SPLINE
SPL {X  -133.930, Y  +759.019, Z    +0.000, E1   +46.142, E3 -160653.483}
SPL {X  -149.331, Y  +728.920, Z    +0.000, E1   +37.154, E3 -160670.653}
SPL {X  -155.856, Y  +707.636, Z    +0.000, E1   +27.210, E3 -160676.656}
SPL {X  -159.260, Y  +686.764, Z    +0.000, E1   +14.026, E3 -160679.931}
SPL {X  -159.985, Y  +672.780, Z    +0.000, E1    +3.059, E3 -160680.832}
SPL {X  -159.990, Y  +669.259, Z    +0.000, E1    -0.225, E3 -160680.888}
SPL {X  -159.990, Y  +665.054, Z    +0.000, E1    -7.292, E3 -160680.993}
SPL {X  -159.990, Y  +658.864, Z    +0.000, E1   -19.708, E3 -160681.381}
SPL {X  -159.990, Y  +650.462, Z    +0.000, E1   -35.240, E3 -160682.392}
SPL {X  -159.990, Y  +636.155, Z    +0.000, E1   -51.890, E3 -160685.290}
SPL {X  -159.990, Y  +583.574, Z    +0.000, E1   -66.740, E3 -160705.086}
SPL {X  -159.990, Y  +451.342, Z    +0.000, E1   -68.591, E3 -160790.778}
ENDSPLINE

SPLINE
SPL {X  -159.990, Y  +495.016, Z    +0.000, E1   -61.398, E3 -160804.742}
ENDSPLINE

SPLINE
SPL {X  -159.990, Y  +469.556, Z    +0.000, E1   -62.943, E3 -160822.182}
SPL {X  -159.990, Y  +452.168, Z    +0.000, E1   -63.738, E3 -160834.737}
SPL {X  -159.990, Y  +433.781, Z    +0.000, E1   -64.535, E3 -160847.762}
SPL {X  -159.990, Y  +407.091, Z    +0.000, E1   -65.705, E3 -160864.966}
SPL {X  -159.990, Y  +383.383, Z    +0.000, E1   -66.590, E3 -160880.100}
SPL {X  -159.086, Y  +365.512, Z    +0.000, E1   -67.201, E3 -160891.198}
SPL {X  -155.924, Y  +346.662, Z    +0.000, E1   -68.026, E3 -160900.715}
SPL {X  -152.004, Y  +332.585, Z    +0.000, E1   -68.049, E3 -160912.153}
SPL {X  -147.728, Y  +321.072, Z    +0.000, E1   -67.490, E3 -160925.735}
SPL {X  -142.939, Y  +310.631, Z    +0.000, E1   -66.808, E3 -160938.802}
SPL {X  -138.502, Y  +302.413, Z    +0.000, E1   -66.138, E3 -160949.544}
SPL {X  -133.815, Y  +294.806, Z    +0.000, E1   -65.413, E3 -160959.751}
SPL {X  -130.038, Y  +289.296, Z    +0.000, E1   -64.749, E3 -160967.342}
SPL {X  -127.114, Y  +285.347, Z    +0.000, E1   -64.250, E3 -160972.765}
SPL {X   -96.237, Y  +254.690, Z    +0.000, E1   -52.223, E3 -161116.153}
ENDSPLINE

SPLINE
SPL {X  -139.640, Y  +304.414, Z    +0.000, E1   -43.367, E3 -161236.514}
SPL {X  -151.122, Y  +329.974, Z    +0.000, E1   -34.701, E3 -161249.306}
SPL {X  -155.699, Y  +345.695, Z    +0.000, E1   -27.167, E3 -161253.687}
SPL {X  -158.589, Y  +361.372, Z    +0.000, E1   -17.765, E3 -161256.451}
SPL {X  -159.702, Y  +372.901, Z    +0.000, E1    -9.563, E3 -161257.683}
SPL {X  -159.980, Y  +380.731, Z    +0.000, E1    -3.359, E3 -161258.081}
SPL {X  -159.990, Y  +384.465, Z    +0.000, E1    -0.049, E3 -161258.138}
SPL {X  -159.990, Y  +385.295, Z    +0.000, E1    +1.130, E3 -161258.144}
SPL {X  -159.990, Y  +387.941, Z    +0.000, E1    +5.453, E3 -161258.208}
SPL {X  -159.990, Y  +392.683, Z    +0.000, E1   +14.335, E3 -161258.465}
SPL {X  -159.990, Y  +399.462, Z    +0.000, E1   +27.551, E3 -161259.151}
SPL {X  -159.990, Y  +406.707, Z    +0.000, E1   +39.277, E3 -161260.307}
SPL {X  -159.990, Y  +418.467, Z    +0.000, E1   +51.591, E3 -161262.913}
SPL {X  -159.990, Y  +469.047, Z    +0.000, E1   +66.225, E3 -161281.990}
SPL {X  -159.990, Y  +610.501, Z    +0.000, E1   +69.067, E3 -161369.594}
SPL {X  -159.990, Y  +630.690, Z    +0.000, E1   +69.080, E3 -161385.974}
SPL {X  -159.990, Y  +652.219, Z    +0.000, E1   +69.078, E3 -161403.459}
SPL {X  -159.990, Y  +671.254, Z    +0.000, E1   +69.063, E3 -161418.959}
SPL {X  -159.471, Y  +684.377, Z    +0.000, E1   +68.989, E3 -161430.187}
SPL {X  -158.115, Y  +695.924, Z    +0.000, E1   +68.836, E3 -161440.970}
SPL {X  -156.463, Y  +704.909, Z    +0.000, E1   +68.615, E3 -161450.028}
SPL {X  -154.598, Y  +712.687, Z    +0.000, E1   +68.393, E3 -161458.242}
SPL {X  -151.859, Y  +721.854, Z    +0.000, E1   +68.046, E3 -161468.461}
SPL {X  -148.628, Y  +730.715, Z    +0.000, E1   +67.614, E3 -161478.870}
SPL {X  -145.416, Y  +738.215, Z    +0.000, E1   +67.166, E3 -161488.078}
SPL {X  -141.128, Y  +746.863, Z    +0.000, E1   +66.582, E3 -161499.055}
SPL {X  -137.485, Y  +753.321, Z    +0.000, E1   +65.984, E3 -161507.632}
SPL {X  -134.819, Y  +757.643, Z    +0.000, E1   +65.575, E3 -161513.427}
SPL {X  -131.187, Y  +763.079, Z    +0.000, E1   +64.994, E3 -161520.810}
SPL {X  -127.405, Y  +768.272, Z    +0.000, E1   +64.349, E3 -161527.931}
SPL {X   -94.830, Y  +800.357, Z    +0.000, E1   +53.815, E3 -161642.463}
ENDSPLINE

SPLINE
SPL {X  -133.930, Y  +759.019, Z    +0.000, E1   +46.142, E3 -161789.846}
SPL {X  -149.331, Y  +728.920, Z    +0.000, E1   +37.154, E3 -161807.017}
SPL {X  -155.856, Y  +707.636, Z    +0.000, E1   +27.210, E3 -161813.020}
SPL {X  -158.677, Y  +691.955, Z    +0.000, E1   +17.570, E3 -161815.726}
SPL {X  -159.802, Y  +679.261, Z    +0.000, E1    +8.330, E3 -161816.922}
SPL {X  -159.990, Y  +669.767, Z    +0.000, E1    +0.394, E3 -161817.247}
SPL {X  -159.990, Y  +667.882, Z    +0.000, E1    -2.380, E3 -161817.269}
SPL {X  -159.990, Y  +664.041, Z    +0.000, E1    -9.423, E3 -161817.395}
SPL {X  -159.990, Y  +660.147, Z    +0.000, E1   -17.275, E3 -161817.632}
SPL {X  -159.990, Y  +656.649, Z    +0.000, E1   -24.355, E3 -161817.939}
SPL {X  -159.990, Y  +650.462, Z    +0.000, E1   -35.240, E3 -161818.756}
SPL {X  -159.990, Y  +636.155, Z    +0.000, E1   -51.890, E3 -161821.653}
SPL {X  -159.990, Y  +583.574, Z    +0.000, E1   -66.740, E3 -161841.450}
SPL {X  -159.990, Y  +451.342, Z    +0.000, E1   -68.591, E3 -161927.141}
ENDSPLINE

SPLINE
SPL {X  -159.990, Y  +495.016, Z    +0.000, E1   -61.398, E3 -161941.106}
ENDSPLINE

SPLINE
SPL {X  -159.990, Y  +469.556, Z    +0.000, E1   -62.943, E3 -161958.545}
SPL {X  -159.990, Y  +445.297, Z    +0.000, E1   -64.051, E3 -161976.035}
SPL {X  -159.990, Y  +420.812, Z    +0.000, E1   -65.111, E3 -161992.625}
SPL {X  -159.990, Y  +395.826, Z    +0.000, E1   -66.138, E3 -162008.561}
SPL {X  -159.536, Y  +370.459, Z    +0.000, E1   -67.052, E3 -162024.454}
SPL {X  -155.924, Y  +346.662, Z    +0.000, E1   -68.026, E3 -162037.079}
SPL {X  -152.004, Y  +332.585, Z    +0.000, E1   -68.049, E3 -162048.517}
SPL {X  -148.519, Y  +323.011, Z    +0.000, E1   -67.572, E3 -162059.794}
SPL {X  -144.736, Y  +314.321, Z    +0.000, E1   -67.058, E3 -162070.491}
SPL {X  -140.646, Y  +306.241, Z    +0.000, E1   -66.458, E3 -162080.870}
SPL {X  -136.388, Y  +298.863, Z    +0.000, E1   -65.814, E3 -162090.642}
SPL {X  -132.805, Y  +293.283, Z    +0.000, E1   -65.214, E3 -162098.232}
SPL {X  -130.038, Y  +289.296, Z    +0.000, E1   -64.749, E3 -162103.706}
SPL {X  -127.114, Y  +285.347, Z    +0.000, E1   -64.250, E3 -162109.129}
SPL {X   -96.237, Y  +254.690, Z    +0.000, E1   -52.223, E3 -162252.517}
ENDSPLINE

SPLINE
SPL {X  -139.640, Y  +304.414, Z    +0.000, E1   -43.367, E3 -162372.878}
SPL {X  -151.122, Y  +329.974, Z    +0.000, E1   -34.701, E3 -162385.670}
SPL {X  -155.699, Y  +345.695, Z    +0.000, E1   -27.167, E3 -162390.051}
SPL {X  -158.589, Y  +361.372, Z    +0.000, E1   -17.765, E3 -162392.815}
SPL {X  -159.702, Y  +372.901, Z    +0.000, E1    -9.563, E3 -162394.047}
SPL {X  -159.980, Y  +380.731, Z    +0.000, E1    -3.359, E3 -162394.445}
SPL {X  -159.990, Y  +384.465, Z    +0.000, E1    -0.049, E3 -162394.502}
SPL {X  -159.990, Y  +386.161, Z    +0.000, E1    +2.359, E3 -162394.525}
SPL {X  -159.990, Y  +391.786, Z    +0.000, E1   +12.382, E3 -162394.775}
SPL {X  -159.990, Y  +399.462, Z    +0.000, E1   +27.551, E3 -162395.515}
SPL {X  -159.990, Y  +406.707, Z    +0.000, E1   +39.277, E3 -162396.671}
SPL {X  -159.990, Y  +418.467, Z    +0.000, E1   +51.591, E3 -162399.276}
SPL {X  -159.990, Y  +469.047, Z    +0.000, E1   +66.225, E3 -162418.354}
SPL {X  -159.990, Y  +610.501, Z    +0.000, E1   +69.067, E3 -162505.957}
SPL {X  -159.990, Y  +623.913, Z    +0.000, E1   +69.046, E3 -162516.906}
SPL {X  -159.990, Y  +635.131, Z    +0.000, E1   +69.053, E3 -162526.007}
SPL {X  -159.990, Y  +652.219, Z    +0.000, E1   +69.078, E3 -162539.822}
SPL {X  -159.990, Y  +671.254, Z    +0.000, E1   +69.063, E3 -162555.323}
SPL {X  -159.471, Y  +684.377, Z    +0.000, E1   +68.989, E3 -162566.550}
SPL {X  -158.115, Y  +695.924, Z    +0.000, E1   +68.836, E3 -162577.334}
SPL {X  -156.463, Y  +704.909, Z    +0.000, E1   +68.615, E3 -162586.391}
SPL {X  -153.837, Y  +715.444, Z    +0.000, E1   +68.325, E3 -162597.569}
SPL {X  -151.088, Y  +724.124, Z    +0.000, E1   +67.925, E3 -162607.479}
SPL {X  -148.628, Y  +730.715, Z    +0.000, E1   +67.614, E3 -162615.234}
SPL {X  -145.416, Y  +738.215, Z    +0.000, E1   +67.166, E3 -162624.442}
SPL {X  -142.090, Y  +745.034, Z    +0.000, E1   +66.692, E3 -162633.098}
SPL {X  -138.343, Y  +751.861, Z    +0.000, E1   +66.137, E3 -162642.025}
SPL {X  -133.893, Y  +759.076, Z    +0.000, E1   +65.453, E3 -162651.701}
SPL {X  -130.341, Y  +764.280, Z    +0.000, E1   +64.831, E3 -162658.839}
SPL {X  -127.405, Y  +768.272, Z    +0.000, E1   +64.349, E3 -162664.294}
SPL {X   -94.830, Y  +800.357, Z    +0.000, E1   +53.815, E3 -162778.827}
ENDSPLINE

SPLINE
SPL {X  -133.930, Y  +759.019, Z    +0.000, E1   +46.142, E3 -162926.210}
SPL {X  -149.331, Y  +728.920, Z    +0.000, E1   +37.154, E3 -162943.381}
SPL {X  -155.856, Y  +707.636, Z    +0.000, E1   +27.210, E3 -162949.384}
SPL {X  -158.677, Y  +691.955, Z    +0.000, E1   +17.570, E3 -162952.090}
SPL {X  -159.802, Y  +679.261, Z    +0.000, E1    +8.330, E3 -162953.286}
SPL {X  -159.990, Y  +671.355, Z    +0.000, E1    +1.732, E3 -162953.596}
SPL {X  -159.990, Y  +669.259, Z    +0.000, E1    -0.225, E3 -162953.615}
SPL {X  -159.990, Y  +665.054, Z    +0.000, E1    -7.292, E3 -162953.720}
SPL {X  -159.990, Y  +658.864, Z    +0.000, E1   -19.708, E3 -162954.108}
SPL {X  -159.990, Y  +650.462, Z    +0.000, E1   -35.240, E3 -162955.120}
SPL {X  -159.990, Y  +636.155, Z    +0.000, E1   -51.890, E3 -162958.017}
SPL {X  -159.990, Y  +583.574, Z    +0.000, E1   -66.740, E3 -162977.813}
SPL {X  -159.990, Y  +451.342, Z    +0.000, E1   -68.591, E3 -163063.505}
ENDSPLINE

SPLINE
SPL {X  -159.990, Y  +495.016, Z    +0.000, E1   -61.398, E3 -163077.470}
ENDSPLINE

SPLINE
SPL {X  -159.990, Y  +473.575, Z    +0.000, E1   -62.704, E3 -163092.204}
SPL {X  -159.990, Y  +455.620, Z    +0.000, E1   -63.615, E3 -163104.822}
SPL {X  -159.990, Y  +433.781, Z    +0.000, E1   -64.535, E3 -163120.490}
SPL {X  -159.990, Y  +414.623, Z    +0.000, E1   -65.374, E3 -163132.910}
SPL {X  -159.990, Y  +395.826, Z    +0.000, E1   -66.138, E3 -163144.924}
SPL {X  -159.536, Y  +370.459, Z    +0.000, E1   -67.052, E3 -163160.817}
SPL {X  -155.924, Y  +346.662, Z    +0.000, E1   -68.026, E3 -163173.442}
SPL {X  -152.751, Y  +334.918, Z    +0.000, E1   -68.124, E3 -163182.272}
SPL {X  -150.185, Y  +327.353, Z    +0.000, E1   -67.790, E3 -163190.995}
SPL {X  -147.824, Y  +321.305, Z    +0.000, E1   -67.459, E3 -163198.258}
SPL {X  -144.736, Y  +314.321, Z    +0.000, E1   -67.058, E3 -163206.854}
SPL {X  -140.646, Y  +306.241, Z    +0.000, E1   -66.458, E3 -163217.233}
SPL {X  -137.570, Y  +300.823, Z    +0.000, E1   -65.968, E3 -163224.425}
SPL {X  -133.815, Y  +294.806, Z    +0.000, E1   -65.413, E3 -163232.478}
SPL {X  -130.038, Y  +289.296, Z    +0.000, E1   -64.749, E3 -163240.070}
SPL {X  -127.114, Y  +285.347, Z    +0.000, E1   -64.250, E3 -163245.493}
SPL {X   -96.237, Y  +254.690, Z    +0.000, E1   -52.223, E3 -163388.881}
ENDSPLINE

SPLINE
SPL {X  -139.640, Y  +304.414, Z    +0.000, E1   -43.367, E3 -163509.242}
SPL {X  -154.086, Y  +339.440, Z    +0.000, E1   -30.439, E3 -163524.799}
SPL {X  -158.589, Y  +361.372, Z    +0.000, E1   -17.765, E3 -163529.179}
SPL {X  -159.702, Y  +372.901, Z    +0.000, E1    -9.563, E3 -163530.411}
SPL {X  -159.980, Y  +380.731, Z    +0.000, E1    -3.359, E3 -163530.808}
SPL {X  -159.990, Y  +384.465, Z    +0.000, E1    -0.049, E3 -163530.866}
SPL {X  -159.990, Y  +386.161, Z    +0.000, E1    +2.359, E3 -163530.888}
SPL {X  -159.990, Y  +391.786, Z    +0.000, E1   +12.382, E3 -163531.139}
SPL {X  -159.990, Y  +399.462, Z    +0.000, E1   +27.551, E3 -163531.879}
SPL {X  -159.990, Y  +406.707, Z    +0.000, E1   +39.277, E3 -163533.034}
SPL {X  -159.990, Y  +418.467, Z    +0.000, E1   +51.591, E3 -163535.640}
SPL {X  -159.990, Y  +469.047, Z    +0.000, E1   +66.225, E3 -163554.717}
SPL {X  -159.990, Y  +610.501, Z    +0.000, E1   +69.067, E3 -163642.321}
SPL {X  -159.990, Y  +630.690, Z    +0.000, E1   +69.080, E3 -163658.701}
SPL {X  -159.990, Y  +648.088, Z    +0.000, E1   +69.056, E3 -163672.878}
SPL {X  -159.990, Y  +663.340, Z    +0.000, E1   +69.061, E3 -163685.264}
SPL {X  -159.706, Y  +681.022, Z    +0.000, E1   +69.040, E3 -163699.896}
SPL {X  -158.115, Y  +695.924, Z    +0.000, E1   +68.836, E3 -163713.697}
SPL {X  -156.463, Y  +704.909, Z    +0.000, E1   +68.615, E3 -163722.755}
SPL {X  -153.837, Y  +715.444, Z    +0.000, E1   +68.325, E3 -163733.932}
SPL {X  -151.088, Y  +724.124, Z    +0.000, E1   +67.925, E3 -163743.843}
SPL {X  -148.628, Y  +730.715, Z    +0.000, E1   +67.614, E3 -163751.597}
SPL {X  -145.416, Y  +738.215, Z    +0.000, E1   +67.166, E3 -163760.806}
SPL {X  -141.128, Y  +746.863, Z    +0.000, E1   +66.582, E3 -163771.783}
SPL {X  -137.485, Y  +753.321, Z    +0.000, E1   +65.984, E3 -163780.359}
SPL {X  -134.819, Y  +757.643, Z    +0.000, E1   +65.575, E3 -163786.154}
SPL {X  -131.187, Y  +763.079, Z    +0.000, E1   +64.994, E3 -163793.538}
SPL {X  -127.405, Y  +768.272, Z    +0.000, E1   +64.349, E3 -163800.658}
SPL {X   -94.830, Y  +800.357, Z    +0.000, E1   +53.815, E3 -163915.190}
ENDSPLINE

SPLINE
SPL {X  -133.930, Y  +759.019, Z    +0.000, E1   +46.142, E3 -164062.574}
SPL {X  -149.331, Y  +728.920, Z    +0.000, E1   +37.154, E3 -164079.744}
SPL {X  -155.856, Y  +707.636, Z    +0.000, E1   +27.210, E3 -164085.747}
SPL {X  -158.677, Y  +691.955, Z    +0.000, E1   +17.570, E3 -164088.453}
SPL {X  -159.802, Y  +679.261, Z    +0.000, E1    +8.330, E3 -164089.650}
SPL {X  -159.990, Y  +671.355, Z    +0.000, E1    +1.732, E3 -164089.960}
SPL {X  -159.990, Y  +669.500, Z    +0.000, E1    +0.000, E3 -164089.977}
SPL {X  -159.990, Y  +667.882, Z    +0.000, E1    -2.380, E3 -164089.996}
SPL {X  -159.990, Y  +664.041, Z    +0.000, E1    -9.423, E3 -164090.122}
SPL {X  -159.990, Y  +658.864, Z    +0.000, E1   -19.708, E3 -164090.472}
SPL {X  -159.990, Y  +650.462, Z    +0.000, E1   -35.240, E3 -164091.483}
SPL {X  -159.990, Y  +636.155, Z    +0.000, E1   -51.890, E3 -164094.381}
SPL {X  -159.990, Y  +583.574, Z    +0.000, E1   -66.740, E3 -164114.177}
SPL {X  -159.990, Y  +451.342, Z    +0.000, E1   -68.591, E3 -164199.869}
ENDSPLINE

SPLINE
SPL {X  -159.990, Y  +495.016, Z    +0.000, E1   -61.398, E3 -164213.833}
ENDSPLINE

SPLINE
SPL {X  -159.990, Y  +473.575, Z    +0.000, E1   -62.704, E3 -164228.568}
SPL {X  -159.990, Y  +455.620, Z    +0.000, E1   -63.615, E3 -164241.186}
SPL {X  -159.990, Y  +433.781, Z    +0.000, E1   -64.535, E3 -164256.853}
SPL {X  -159.990, Y  +407.091, Z    +0.000, E1   -65.705, E3 -164274.057}
SPL {X  -159.990, Y  +383.383, Z    +0.000, E1   -66.590, E3 -164289.191}
SPL {X  -158.268, Y  +359.089, Z    +0.000, E1   -67.514, E3 -164303.392}
SPL {X  -153.587, Y  +337.689, Z    +0.000, E1   -68.173, E3 -164316.126}
SPL {X  -150.185, Y  +327.353, Z    +0.000, E1   -67.790, E3 -164327.358}
SPL {X  -147.824, Y  +321.305, Z    +0.000, E1   -67.459, E3 -164334.622}
SPL {X  -144.736, Y  +314.321, Z    +0.000, E1   -67.058, E3 -164343.218}
SPL {X  -140.646, Y  +306.241, Z    +0.000, E1   -66.458, E3 -164353.597}
SPL {X  -136.388, Y  +298.863, Z    +0.000, E1   -65.814, E3 -164363.370}
SPL {X  -132.805, Y  +293.283, Z    +0.000, E1   -65.214, E3 -164370.959}
SPL {X  -130.038, Y  +289.296, Z    +0.000, E1   -64.749, E3 -164376.433}
SPL {X  -127.114, Y  +285.347, Z    +0.000, E1   -64.250, E3 -164381.856}
SPL {X   -96.237, Y  +254.690, Z    +0.000, E1   -52.223, E3 -164525.244}
ENDSPLINE

SPLINE
SPL {X  -139.640, Y  +304.414, Z    +0.000, E1   -43.367, E3 -164645.605}
SPL {X  -154.086, Y  +339.440, Z    +0.000, E1   -30.439, E3 -164661.162}
SPL {X  -158.589, Y  +361.372, Z    +0.000, E1   -17.765, E3 -164665.542}
SPL {X  -159.702, Y  +372.901, Z    +0.000, E1    -9.563, E3 -164666.774}
SPL {X  -159.980, Y  +380.731, Z    +0.000, E1    -3.359, E3 -164667.172}
SPL {X  -159.990, Y  +384.465, Z    +0.000, E1    -0.049, E3 -164667.229}
SPL {X  -159.990, Y  +386.161, Z    +0.000, E1    +2.359, E3 -164667.252}
SPL {X  -159.990, Y  +390.716, Z    +0.000, E1   +10.524, E3 -164667.427}
SPL {X  -159.990, Y  +397.792, Z    +0.000, E1   +24.215, E3 -164668.057}
SPL {X  -159.990, Y  +406.707, Z    +0.000, E1   +39.277, E3 -164669.398}
SPL {X  -159.990, Y  +418.467, Z    +0.000, E1   +51.591, E3 -164672.004}
SPL {X  -159.990, Y  +469.047, Z    +0.000, E1   +66.225, E3 -164691.081}
SPL {X  -159.990, Y  +610.501, Z    +0.000, E1   +69.067, E3 -164778.685}
SPL {X  -159.990, Y  +630.690, Z    +0.000, E1   +69.080, E3 -164795.065}
SPL {X  -159.990, Y  +652.219, Z    +0.000, E1   +69.078, E3 -164812.550}
SPL {X  -159.990, Y  +671.254, Z    +0.000, E1   +69.063, E3 -164828.050}
SPL {X  -159.172, Y  +687.655, Z    +0.000, E1   +68.973, E3 -164842.210}
SPL {X  -157.106, Y  +701.739, Z    +0.000, E1   +68.720, E3 -164855.818}
SPL {X  -153.837, Y  +715.444, Z    +0.000, E1   +68.325, E3 -164870.296}
SPL {X  -151.088, Y  +724.124, Z    +0.000, E1   +67.925, E3 -164880.206}
SPL {X  -148.628, Y  +730.715, Z    +0.000, E1   +67.614, E3 -164887.961}
SPL {X  -145.416, Y  +738.215, Z    +0.000, E1   +67.166, E3 -164897.169}
SPL {X  -142.090, Y  +745.034, Z    +0.000, E1   +66.692, E3 -164905.825}
SPL {X  -138.343, Y  +751.861, Z    +0.000, E1   +66.137, E3 -164914.752}
SPL {X  -133.893, Y  +759.076, Z    +0.000, E1   +65.453, E3 -164924.428}
SPL {X  -130.341, Y  +764.280, Z    +0.000, E1   +64.831, E3 -164931.566}
SPL {X  -127.405, Y  +768.272, Z    +0.000, E1   +64.349, E3 -164937.022}
SPL {X   -94.830, Y  +800.357, Z    +0.000, E1   +53.815, E3 -165051.554}
ENDSPLINE

SPLINE
SPL {X  -133.930, Y  +759.019, Z    +0.000, E1   +46.142, E3 -165198.937}
SPL {X  -149.331, Y  +728.920, Z    +0.000, E1   +37.154, E3 -165216.108}
SPL {X  -155.856, Y  +707.636, Z    +0.000, E1   +27.210, E3 -165222.111}
SPL {X  -158.677, Y  +691.955, Z    +0.000, E1   +17.570, E3 -165224.817}
SPL {X  -159.802, Y  +679.261, Z    +0.000, E1    +8.330, E3 -165226.013}
SPL {X  -159.990, Y  +669.483, Z    +0.000, E1    +0.154, E3 -165226.340}
SPL {X  -159.990, Y  +665.054, Z    +0.000, E1    -7.292, E3 -165226.447}
SPL {X  -159.990, Y  +660.147, Z    +0.000, E1   -17.275, E3 -165226.723}
SPL {X  -159.990, Y  +656.649, Z    +0.000, E1   -24.355, E3 -165227.030}
SPL {X  -159.990, Y  +650.462, Z    +0.000, E1   -35.240, E3 -165227.847}
SPL {X  -159.990, Y  +636.155, Z    +0.000, E1   -51.890, E3 -165230.744}
SPL {X  -159.990, Y  +583.574, Z    +0.000, E1   -66.740, E3 -165250.541}
SPL {X  -159.990, Y  +451.342, Z    +0.000, E1   -68.591, E3 -165336.232}
ENDSPLINE

SPLINE
SPL {X  -159.990, Y  +495.016, Z    +0.000, E1   -61.398, E3 -165350.197}
ENDSPLINE

SPLINE
SPL {X  -159.990, Y  +473.575, Z    +0.000, E1   -62.704, E3 -165364.932}
SPL {X  -159.990, Y  +455.620, Z    +0.000, E1   -63.615, E3 -165377.550}
SPL {X  -159.990, Y  +433.781, Z    +0.000, E1   -64.535, E3 -165393.217}
SPL {X  -159.990, Y  +414.623, Z    +0.000, E1   -65.374, E3 -165405.637}
SPL {X  -159.990, Y  +395.826, Z    +0.000, E1   -66.138, E3 -165417.652}
SPL {X  -159.536, Y  +370.459, Z    +0.000, E1   -67.052, E3 -165433.544}
SPL {X  -155.924, Y  +346.662, Z    +0.000, E1   -68.026, E3 -165446.170}
SPL {X  -152.751, Y  +334.918, Z    +0.000, E1   -68.124, E3 -165455.000}
SPL {X  -150.185, Y  +327.353, Z    +0.000, E1   -67.790, E3 -165463.722}
SPL {X  -147.824, Y  +321.305, Z    +0.000, E1   -67.459, E3 -165470.985}
SPL {X  -144.736, Y  +314.321, Z    +0.000, E1   -67.058, E3 -165479.582}
SPL {X  -140.646, Y  +306.241, Z    +0.000, E1   -66.458, E3 -165489.961}
SPL {X  -137.570, Y  +300.823, Z    +0.000, E1   -65.968, E3 -165497.152}
SPL {X  -133.815, Y  +294.806, Z    +0.000, E1   -65.413, E3 -165505.205}
SPL {X  -130.038, Y  +289.296, Z    +0.000, E1   -64.749, E3 -165512.797}
SPL {X  -127.114, Y  +285.347, Z    +0.000, E1   -64.250, E3 -165518.220}
SPL {X   -96.237, Y  +254.690, Z    +0.000, E1   -52.223, E3 -165661.608}
ENDSPLINE

SPLINE
SPL {X  -139.640, Y  +304.414, Z    +0.000, E1   -43.367, E3 -165781.969}
SPL {X  -154.086, Y  +339.440, Z    +0.000, E1   -30.439, E3 -165797.526}
SPL {X  -158.589, Y  +361.372, Z    +0.000, E1   -17.765, E3 -165801.906}
SPL {X  -159.702, Y  +372.901, Z    +0.000, E1    -9.563, E3 -165803.138}
SPL {X  -159.980, Y  +380.731, Z    +0.000, E1    -3.359, E3 -165803.536}
SPL {X  -159.990, Y  +384.708, Z    +0.000, E1    +0.166, E3 -165803.595}
SPL {X  -159.990, Y  +387.941, Z    +0.000, E1    +5.453, E3 -165803.662}
SPL {X  -159.990, Y  +391.582, Z    +0.000, E1   +12.331, E3 -165803.837}
SPL {X  -159.990, Y  +397.792, Z    +0.000, E1   +24.215, E3 -165804.421}
SPL {X  -159.990, Y  +406.707, Z    +0.000, E1   +39.277, E3 -165805.762}
SPL {X  -159.990, Y  +418.467, Z    +0.000, E1   +51.591, E3 -165808.367}
SPL {X  -159.990, Y  +469.047, Z    +0.000, E1   +66.225, E3 -165827.444}
SPL {X  -159.990, Y  +610.501, Z    +0.000, E1   +69.067, E3 -165915.048}
SPL {X  -159.990, Y  +630.690, Z    +0.000, E1   +69.080, E3 -165931.429}
SPL {X  -159.990, Y  +648.088, Z    +0.000, E1   +69.056, E3 -165945.605}
SPL {X  -159.990, Y  +663.340, Z    +0.000, E1   +69.061, E3 -165957.991}
SPL {X  -159.706, Y  +681.022, Z    +0.000, E1   +69.040, E3 -165972.624}
SPL {X  -158.115, Y  +695.924, Z    +0.000, E1   +68.836, E3 -165986.425}
SPL {X  -156.463, Y  +704.909, Z    +0.000, E1   +68.615, E3 -165995.482}
SPL {X  -153.837, Y  +715.444, Z    +0.000, E1   +68.325, E3 -166006.660}
SPL {X  -151.088, Y  +724.124, Z    +0.000, E1   +67.925, E3 -166016.570}
SPL {X  -148.628, Y  +730.715, Z    +0.000, E1   +67.614, E3 -166024.325}
SPL {X  -145.416, Y  +738.215, Z    +0.000, E1   +67.166, E3 -166033.533}
SPL {X  -142.090, Y  +745.034, Z    +0.000, E1   +66.692, E3 -166042.189}
SPL {X  -138.343, Y  +751.861, Z    +0.000, E1   +66.137, E3 -166051.115}
SPL {X  -133.893, Y  +759.076, Z    +0.000, E1   +65.453, E3 -166060.791}
SPL {X  -130.341, Y  +764.280, Z    +0.000, E1   +64.831, E3 -166067.930}
SPL {X  -127.405, Y  +768.272, Z    +0.000, E1   +64.349, E3 -166073.385}
SPL {X   -94.830, Y  +800.357, Z    +0.000, E1   +53.815, E3 -166187.917}
ENDSPLINE

SPLINE
SPL {X  -133.930, Y  +759.019, Z    +0.000, E1   +46.142, E3 -166335.301}
SPL {X  -149.331, Y  +728.920, Z    +0.000, E1   +37.154, E3 -166352.471}
SPL {X  -155.856, Y  +707.636, Z    +0.000, E1   +27.210, E3 -166358.475}
SPL {X  -159.260, Y  +686.764, Z    +0.000, E1   +14.026, E3 -166361.749}
SPL {X  -159.985, Y  +672.780, Z    +0.000, E1    +3.059, E3 -166362.650}
SPL {X  -159.990, Y  +669.259, Z    +0.000, E1    -0.225, E3 -166362.706}
SPL {X  -159.990, Y  +665.054, Z    +0.000, E1    -7.292, E3 -166362.811}
SPL {X  -159.990, Y  +658.864, Z    +0.000, E1   -19.708, E3 -166363.199}
SPL {X  -159.990, Y  +650.462, Z    +0.000, E1   -35.240, E3 -166364.211}
SPL {X  -159.990, Y  +636.155, Z    +0.000, E1   -51.890, E3 -166367.108}
SPL {X  -159.990, Y  +583.574, Z    +0.000, E1   -66.740, E3 -166386.904}
SPL {X  -159.990, Y  +451.342, Z    +0.000, E1   -68.591, E3 -166472.596}
ENDSPLINE

SPLINE
SPL {X  -159.990, Y  +495.016, Z    +0.000, E1   -61.398, E3 -166486.561}
ENDSPLINE

SPLINE
SPL {X  -159.990, Y  +469.556, Z    +0.000, E1   -62.943, E3 -166504.000}
SPL {X  -159.990, Y  +445.297, Z    +0.000, E1   -64.051, E3 -166521.489}
SPL {X  -159.990, Y  +420.812, Z    +0.000, E1   -65.111, E3 -166538.080}
SPL {X  -159.990, Y  +395.826, Z    +0.000, E1   -66.138, E3 -166554.015}
SPL {X  -159.536, Y  +370.459, Z    +0.000, E1   -67.052, E3 -166569.908}
SPL {X  -157.113, Y  +352.293, Z    +0.000, E1   -67.811, E3 -166579.490}
SPL {X  -153.587, Y  +337.689, Z    +0.000, E1   -68.173, E3 -166588.853}
SPL {X  -150.185, Y  +327.353, Z    +0.000, E1   -67.790, E3 -166600.086}
SPL {X  -147.050, Y  +319.468, Z    +0.000, E1   -67.370, E3 -166609.566}
SPL {X  -142.939, Y  +310.631, Z    +0.000, E1   -66.808, E3 -166620.620}
SPL {X  -138.502, Y  +302.413, Z    +0.000, E1   -66.138, E3 -166631.363}
SPL {X  -135.296, Y  +297.108, Z    +0.000, E1   -65.610, E3 -166638.502}
SPL {X  -132.805, Y  +293.283, Z    +0.000, E1   -65.214, E3 -166643.686}
SPL {X  -130.038, Y  +289.296, Z    +0.000, E1   -64.749, E3 -166649.160}
SPL {X  -127.114, Y  +285.347, Z    +0.000, E1   -64.250, E3 -166654.583}
SPL {X   -96.237, Y  +254.690, Z    +0.000, E1   -52.223, E3 -166797.972}
ENDSPLINE

SPLINE
SPL {X  -139.640, Y  +304.414, Z    +0.000, E1   -43.367, E3 -166918.332}
SPL {X  -154.086, Y  +339.440, Z    +0.000, E1   -30.439, E3 -166933.890}
SPL {X  -158.589, Y  +361.372, Z    +0.000, E1   -17.765, E3 -166938.270}
SPL {X  -159.702, Y  +372.901, Z    +0.000, E1    -9.563, E3 -166939.501}
SPL {X  -159.980, Y  +380.731, Z    +0.000, E1    -3.359, E3 -166939.899}
SPL {X  -159.990, Y  +384.465, Z    +0.000, E1    -0.049, E3 -166939.957}
SPL {X  -159.990, Y  +386.161, Z    +0.000, E1    +2.359, E3 -166939.979}
SPL {X  -159.990, Y  +391.786, Z    +0.000, E1   +12.382, E3 -166940.230}
SPL {X  -159.990, Y  +399.462, Z    +0.000, E1   +27.551, E3 -166940.970}
SPL {X  -159.990, Y  +406.707, Z    +0.000, E1   +39.277, E3 -166942.125}
SPL {X  -159.990, Y  +418.467, Z    +0.000, E1   +51.591, E3 -166944.731}
SPL {X  -159.990, Y  +469.047, Z    +0.000, E1   +66.225, E3 -166963.808}
SPL {X  -159.990, Y  +610.501, Z    +0.000, E1   +69.067, E3 -167051.412}
SPL {X  -159.990, Y  +630.690, Z    +0.000, E1   +69.080, E3 -167067.792}
SPL {X  -159.990, Y  +648.088, Z    +0.000, E1   +69.056, E3 -167081.969}
SPL {X  -159.990, Y  +663.340, Z    +0.000, E1   +69.061, E3 -167094.355}
SPL {X  -159.706, Y  +681.022, Z    +0.000, E1   +69.040, E3 -167108.987}
SPL {X  -158.115, Y  +695.924, Z    +0.000, E1   +68.836, E3 -167122.788}
SPL {X  -156.463, Y  +704.909, Z    +0.000, E1   +68.615, E3 -167131.846}
SPL {X  -153.837, Y  +715.444, Z    +0.000, E1   +68.325, E3 -167143.023}
SPL {X  -151.088, Y  +724.124, Z    +0.000, E1   +67.925, E3 -167152.933}
SPL {X  -148.628, Y  +730.715, Z    +0.000, E1   +67.614, E3 -167160.688}
SPL {X  -145.416, Y  +738.215, Z    +0.000, E1   +67.166, E3 -167169.897}
SPL {X  -141.128, Y  +746.863, Z    +0.000, E1   +66.582, E3 -167180.874}
SPL {X  -137.485, Y  +753.321, Z    +0.000, E1   +65.984, E3 -167189.450}
SPL {X  -134.819, Y  +757.643, Z    +0.000, E1   +65.575, E3 -167195.245}
SPL {X  -131.187, Y  +763.079, Z    +0.000, E1   +64.994, E3 -167202.628}
SPL {X  -127.405, Y  +768.272, Z    +0.000, E1   +64.349, E3 -167209.749}
SPL {X   -94.830, Y  +800.357, Z    +0.000, E1   +53.815, E3 -167324.281}
ENDSPLINE

SPLINE
SPL {X  -133.930, Y  +759.019, Z    +0.000, E1   +46.142, E3 -167471.665}
SPL {X  -149.331, Y  +728.920, Z    +0.000, E1   +37.154, E3 -167488.835}
SPL {X  -155.856, Y  +707.636, Z    +0.000, E1   +27.210, E3 -167494.838}
SPL {X  -158.677, Y  +691.955, Z    +0.000, E1   +17.570, E3 -167497.544}
SPL {X  -159.802, Y  +679.261, Z    +0.000, E1    +8.330, E3 -167498.741}
SPL {X  -159.990, Y  +671.355, Z    +0.000, E1    +1.732, E3 -167499.050}
SPL {X  -159.990, Y  +669.500, Z    +0.000, E1    +0.000, E3 -167499.068}
SPL {X  -159.990, Y  +667.882, Z    +0.000, E1    -2.380, E3 -167499.087}
SPL {X  -159.990, Y  +664.041, Z    +0.000, E1    -9.423, E3 -167499.213}
SPL {X  -159.990, Y  +658.864, Z    +0.000, E1   -19.708, E3 -167499.563}
SPL {X  -159.990, Y  +650.462, Z    +0.000, E1   -35.240, E3 -167500.574}
SPL {X  -159.990, Y  +636.155, Z    +0.000, E1   -51.890, E3 -167503.472}
SPL {X  -159.990, Y  +583.574, Z    +0.000, E1   -66.740, E3 -167523.268}
SPL {X  -159.990, Y  +451.342, Z    +0.000, E1   -68.591, E3 -167608.960}
ENDSPLINE

SPLINE
SPL {X  -159.990, Y  +501.364, Z    +0.000, E1   -60.990, E3 -167618.270}
ENDSPLINE

SPLINE
SPL {X  -159.990, Y  +489.357, Z    +0.000, E1   -61.712, E3 -167627.113}
SPL {X  -159.990, Y  +473.575, Z    +0.000, E1   -62.704, E3 -167637.659}
SPL {X  -159.990, Y  +455.620, Z    +0.000, E1   -63.615, E3 -167650.277}
SPL {X  -159.990, Y  +439.579, Z    +0.000, E1   -64.263, E3 -167662.012}
SPL {X  -159.990, Y  +420.812, Z    +0.000, E1   -65.111, E3 -167674.444}
SPL {X  -159.990, Y  +395.826, Z    +0.000, E1   -66.138, E3 -167690.379}
SPL {X  -159.536, Y  +370.459, Z    +0.000, E1   -67.052, E3 -167706.272}
SPL {X  -155.899, Y  +346.553, Z    +0.000, E1   -68.023, E3 -167719.018}
SPL {X  -155.470, Y  +344.740, Z    +0.000, E1   -66.275, E3 -167734.431}
SPL {X  -151.958, Y  +332.444, Z    +0.000, E1   -65.791, E3 -167749.177}
SPL {X  -148.012, Y  +321.760, Z    +0.000, E1   -65.212, E3 -167762.811}
SPL {X  -144.181, Y  +313.155, Z    +0.000, E1   -64.628, E3 -167774.320}
SPL {X  -141.300, Y  +307.460, Z    +0.000, E1   -64.150, E3 -167782.212}
SPL {X  -138.693, Y  +302.744, Z    +0.000, E1   -63.741, E3 -167788.826}
SPL {X  -135.031, Y  +296.690, Z    +0.000, E1   -63.147, E3 -167797.488}
SPL {X  -130.494, Y  +289.936, Z    +0.000, E1   -62.364, E3 -167807.326}
SPL {X  -102.192, Y  +259.400, Z    +0.000, E1   -52.167, E3 -167926.050}
ENDSPLINE

SPLINE
SPL {X  -140.725, Y  +306.386, Z    +0.000, E1   -41.058, E3 -168050.944}
SPL {X  -153.851, Y  +338.606, Z    +0.000, E1   -29.149, E3 -168067.561}
SPL {X  -158.264, Y  +359.064, Z    +0.000, E1   -18.155, E3 -168072.512}
SPL {X  -159.641, Y  +371.933, Z    +0.000, E1    -9.693, E3 -168074.247}
SPL {X  -159.986, Y  +381.420, Z    +0.000, E1    -2.704, E3 -168074.813}
SPL {X  -159.990, Y  +384.527, Z    +0.000, E1    +0.013, E3 -168074.873}
SPL {X  -159.990, Y  +386.984, Z    +0.000, E1    +3.187, E3 -168074.925}
SPL {X  -159.990, Y  +392.544, Z    +0.000, E1   +12.471, E3 -168075.238}
SPL {X  -159.990, Y  +397.827, Z    +0.000, E1   +22.184, E3 -168075.759}
SPL {X  -159.990, Y  +403.857, Z    +0.000, E1   +31.979, E3 -168076.723}
SPL {X  -159.990, Y  +417.858, Z    +0.000, E1   +47.695, E3 -168080.208}
SPL {X  -159.990, Y  +475.808, Z    +0.000, E1   +64.751, E3 -168104.162}
SPL {X  -159.990, Y  +590.266, Z    +0.000, E1   +66.680, E3 -168187.279}
SPL {X  -159.990, Y  +611.678, Z    +0.000, E1   +66.672, E3 -168206.919}
SPL {X  -159.990, Y  +629.811, Z    +0.000, E1   +66.653, E3 -168223.575}
SPL {X  -159.990, Y  +646.024, Z    +0.000, E1   +66.650, E3 -168238.451}
SPL {X  -159.990, Y  +658.527, Z    +0.000, E1   +66.634, E3 -168249.933}
SPL {X  -159.990, Y  +671.049, Z    +0.000, E1   +66.648, E3 -168261.382}
SPL {X  -159.584, Y  +682.893, Z    +0.000, E1   +66.583, E3 -168272.679}
SPL {X  -158.332, Y  +694.472, Z    +0.000, E1   +66.450, E3 -168284.553}
SPL {X  -156.148, Y  +706.350, Z    +0.000, E1   +66.133, E3 -168297.764}
SPL {X  -154.052, Y  +714.685, Z    +0.000, E1   +65.842, E3 -168307.551}
SPL {X  -151.974, Y  +721.507, Z    +0.000, E1   +65.548, E3 -168315.908}
SPL {X  -149.510, Y  +728.452, Z    +0.000, E1   +65.197, E3 -168324.751}
SPL {X  -145.784, Y  +737.407, Z    +0.000, E1   +64.671, E3 -168336.542}
SPL {X  -142.587, Y  +744.066, Z    +0.000, E1   +64.133, E3 -168345.725}
SPL {X  -139.326, Y  +750.145, Z    +0.000, E1   +63.650, E3 -168354.218}
SPL {X  -135.791, Y  +756.103, Z    +0.000, E1   +63.018, E3 -168362.863}
SPL {X  -133.172, Y  +760.168, Z    +0.000, E1   +62.565, E3 -168368.788}
SPL {X  -130.070, Y  +764.659, Z    +0.000, E1   +62.024, E3 -168375.383}
SPL {X  -103.420, Y  +793.570, Z    +0.000, E1   +51.337, E3 -168505.283}
ENDSPLINE

SPLINE
SPL {X  -132.256, Y  +761.529, Z    +0.000, E1   +44.935, E3 -168611.373}
SPL {X  -148.790, Y  +730.309, Z    +0.000, E1   +35.907, E3 -168632.646}
SPL {X  -157.132, Y  +701.603, Z    +0.000, E1   +22.438, E3 -168641.907}
SPL {X  -159.426, Y  +684.927, Z    +0.000, E1   +11.876, E3 -168644.526}
SPL {X  -159.929, Y  +675.915, Z    +0.000, E1    +5.290, E3 -168645.237}
SPL {X  -159.990, Y  +669.794, Z    +0.000, E1    +0.371, E3 -168645.410}
SPL {X  -159.990, Y  +668.338, Z    +0.000, E1    -1.468, E3 -168645.427}
SPL {X  -159.990, Y  +665.597, Z    +0.000, E1    -5.793, E3 -168645.505}
SPL {X  -159.990, Y  +662.769, Z    +0.000, E1   -10.720, E3 -168645.657}
SPL {X  -159.990, Y  +658.787, Z    +0.000, E1   -17.995, E3 -168645.985}
SPL {X  -159.990, Y  +653.215, Z    +0.000, E1   -27.908, E3 -168646.677}
SPL {X  -159.990, Y  +646.194, Z    +0.000, E1   -38.517, E3 -168647.965}
SPL {X  -159.990, Y  +636.314, Z    +0.000, E1   -48.490, E3 -168650.603}
SPL {X  -159.990, Y  +588.081, Z    +0.000, E1   -63.406, E3 -168671.785}
SPL {X  -159.990, Y  +471.514, Z    +0.000, E1   -66.231, E3 -168755.293}
SPL {X  -159.990, Y  +458.012, Z    +0.000, E1   -66.224, E3 -168767.922}
SPL {X  -159.990, Y  +445.900, Z    +0.000, E1   -66.225, E3 -168779.235}
ENDSPLINE

SPLINE
SPL {X  -159.990, Y  +468.953, Z    +0.000, E1   -61.697, E3 -168789.194}
ENDSPLINE

SPLINE
SPL {X  -159.990, Y  +457.098, Z    +0.000, E1   -61.912, E3 -168801.290}
SPL {X  -159.990, Y  +442.075, Z    +0.000, E1   -62.596, E3 -168813.066}
SPL {X  -159.990, Y  +430.868, Z    +0.000, E1   -63.135, E3 -168821.319}
SPL {X  -159.990, Y  +416.857, Z    +0.000, E1   -63.835, E3 -168830.986}
SPL {X  -159.990, Y  +402.942, Z    +0.000, E1   -64.377, E3 -168841.215}
SPL {X  -159.990, Y  +382.745, Z    +0.000, E1   -65.209, E3 -168855.129}
SPL {X  -158.929, Y  +364.101, Z    +0.000, E1   -65.981, E3 -168866.884}
SPL {X  -156.693, Y  +350.188, Z    +0.000, E1   -66.345, E3 -168877.008}
SPL {X  -154.578, Y  +341.238, Z    +0.000, E1   -66.113, E3 -168886.766}
SPL {X  -151.958, Y  +332.444, Z    +0.000, E1   -65.791, E3 -168897.326}
SPL {X  -148.012, Y  +321.760, Z    +0.000, E1   -65.212, E3 -168910.959}
SPL {X  -145.172, Y  +315.256, Z    +0.000, E1   -64.753, E3 -168919.664}
SPL {X  -142.205, Y  +309.188, Z    +0.000, E1   -64.322, E3 -168927.917}
SPL {X  -138.693, Y  +302.744, Z    +0.000, E1   -63.741, E3 -168936.974}
SPL {X  -135.977, Y  +298.197, Z    +0.000, E1   -63.280, E3 -168943.494}
SPL {X  -132.828, Y  +293.318, Z    +0.000, E1   -62.759, E3 -168950.548}
SPL {X  -129.451, Y  +288.482, Z    +0.000, E1   -62.137, E3 -168957.651}
SPL {X  -102.192, Y  +259.400, Z    +0.000, E1   -52.167, E3 -169074.198}
ENDSPLINE

SPLINE
SPL {X  -140.725, Y  +306.386, Z    +0.000, E1   -41.058, E3 -169199.092}
SPL {X  -153.851, Y  +338.606, Z    +0.000, E1   -29.149, E3 -169215.709}
SPL {X  -158.264, Y  +359.064, Z    +0.000, E1   -18.155, E3 -169220.660}
SPL {X  -159.641, Y  +371.933, Z    +0.000, E1    -9.693, E3 -169222.396}
SPL {X  -159.986, Y  +381.420, Z    +0.000, E1    -2.704, E3 -169222.961}
SPL {X  -159.990, Y  +384.527, Z    +0.000, E1    +0.013, E3 -169223.021}
SPL {X  -159.990, Y  +385.909, Z    +0.000, E1    +1.800, E3 -169223.039}
SPL {X  -159.990, Y  +389.230, Z    +0.000, E1    +6.815, E3 -169223.163}
SPL {X  -159.990, Y  +395.332, Z    +0.000, E1   +17.451, E3 -169223.646}
SPL {X  -159.990, Y  +403.857, Z    +0.000, E1   +31.979, E3 -169224.871}
SPL {X  -159.990, Y  +417.858, Z    +0.000, E1   +47.695, E3 -169228.356}
SPL {X  -159.990, Y  +475.808, Z    +0.000, E1   +64.751, E3 -169252.310}
SPL {X  -159.990, Y  +590.266, Z    +0.000, E1   +66.680, E3 -169335.427}
SPL {X  -159.990, Y  +605.903, Z    +0.000, E1   +66.635, E3 -169349.846}
SPL {X  -159.990, Y  +620.525, Z    +0.000, E1   +66.669, E3 -169363.180}
SPL {X  -159.990, Y  +638.202, Z    +0.000, E1   +66.649, E3 -169379.430}
SPL {X  -159.990, Y  +654.774, Z    +0.000, E1   +66.658, E3 -169394.599}
SPL {X  -159.990, Y  +671.049, Z    +0.000, E1   +66.648, E3 -169409.530}
SPL {X  -159.584, Y  +682.893, Z    +0.000, E1   +66.583, E3 -169420.827}
SPL {X  -158.845, Y  +690.607, Z    +0.000, E1   +66.486, E3 -169428.680}
SPL {X  -157.279, Y  +700.830, Z    +0.000, E1   +66.296, E3 -169439.661}
SPL {X  -154.589, Y  +712.719, Z    +0.000, E1   +65.941, E3 -169453.304}
SPL {X  -151.974, Y  +721.507, Z    +0.000, E1   +65.548, E3 -169464.056}
SPL {X  -149.510, Y  +728.452, Z    +0.000, E1   +65.197, E3 -169472.899}
SPL {X  -146.809, Y  +735.092, Z    +0.000, E1   +64.789, E3 -169481.646}
SPL {X  -143.550, Y  +742.141, Z    +0.000, E1   +64.312, E3 -169491.165}
SPL {X  -140.309, Y  +748.378, Z    +0.000, E1   +63.779, E3 -169499.898}
SPL {X  -136.621, Y  +754.755, Z    +0.000, E1   +63.190, E3 -169509.015}
SPL {X  -133.172, Y  +760.168, Z    +0.000, E1   +62.565, E3 -169516.936}
SPL {X  -130.070, Y  +764.659, Z    +0.000, E1   +62.024, E3 -169523.531}
SPL {X  -103.420, Y  +793.570, Z    +0.000, E1   +51.337, E3 -169653.431}
ENDSPLINE

SPLINE
SPL {X  -141.359, Y  +746.429, Z    +0.000, E1   +41.207, E3 -169771.645}
SPL {X  -153.791, Y  +715.605, Z    +0.000, E1   +29.700, E3 -169786.414}
SPL {X  -157.923, Y  +697.131, Z    +0.000, E1   +19.758, E3 -169790.946}
SPL {X  -159.426, Y  +684.927, Z    +0.000, E1   +11.876, E3 -169792.674}
SPL {X  -159.929, Y  +675.915, Z    +0.000, E1    +5.290, E3 -169793.385}
SPL {X  -159.990, Y  +669.794, Z    +0.000, E1    +0.371, E3 -169793.558}
SPL {X  -159.990, Y  +668.338, Z    +0.000, E1    -1.468, E3 -169793.575}
SPL {X  -159.990, Y  +664.217, Z    +0.000, E1    -7.944, E3 -169793.727}
SPL {X  -159.990, Y  +657.963, Z    +0.000, E1   -19.417, E3 -169794.224}
SPL {X  -159.990, Y  +649.570, Z    +0.000, E1   -33.681, E3 -169795.448}
SPL {X  -159.990, Y  +636.314, Z    +0.000, E1   -48.490, E3 -169798.751}
SPL {X  -159.990, Y  +588.081, Z    +0.000, E1   -63.406, E3 -169819.933}
SPL {X  -159.990, Y  +471.514, Z    +0.000, E1   -66.231, E3 -169903.441}
SPL {X  -159.990, Y  +458.012, Z    +0.000, E1   -66.224, E3 -169916.070}
SPL {X  -159.990, Y  +445.900, Z    +0.000, E1   -66.225, E3 -169927.383}
ENDSPLINE

SPLINE
SPL {X  -159.990, Y  +465.730, Z    +0.000, E1   -61.693, E3 -169941.208}
ENDSPLINE

SPLINE
SPL {X  -159.990, Y  +446.910, Z    +0.000, E1   -62.394, E3 -169957.428}
SPL {X  -159.990, Y  +430.868, Z    +0.000, E1   -63.135, E3 -169969.467}
SPL {X  -159.990, Y  +416.857, Z    +0.000, E1   -63.835, E3 -169979.134}
SPL {X  -159.990, Y  +402.942, Z    +0.000, E1   -64.377, E3 -169989.363}
SPL {X  -159.990, Y  +382.745, Z    +0.000, E1   -65.209, E3 -170003.277}
SPL {X  -158.342, Y  +359.598, Z    +0.000, E1   -66.150, E3 -170017.982}
SPL {X  -155.453, Y  +344.669, Z    +0.000, E1   -66.270, E3 -170030.824}
SPL {X  -151.958, Y  +332.444, Z    +0.000, E1   -65.791, E3 -170045.474}
SPL {X  -148.012, Y  +321.760, Z    +0.000, E1   -65.212, E3 -170059.107}
SPL {X  -144.181, Y  +313.155, Z    +0.000, E1   -64.628, E3 -170070.617}
SPL {X  -141.300, Y  +307.460, Z    +0.000, E1   -64.150, E3 -170078.508}
SPL {X  -138.693, Y  +302.744, Z    +0.000, E1   -63.741, E3 -170085.122}
SPL {X  -135.031, Y  +296.690, Z    +0.000, E1   -63.147, E3 -170093.784}
SPL {X  -130.494, Y  +289.936, Z    +0.000, E1   -62.364, E3 -170103.622}
SPL {X  -102.192, Y  +259.400, Z    +0.000, E1   -52.167, E3 -170222.346}
ENDSPLINE

SPLINE
SPL {X  -140.725, Y  +306.386, Z    +0.000, E1   -41.058, E3 -170347.240}
SPL {X  -153.851, Y  +338.606, Z    +0.000, E1   -29.149, E3 -170363.857}
SPL {X  -158.264, Y  +359.064, Z    +0.000, E1   -18.155, E3 -170368.809}
SPL {X  -159.641, Y  +371.933, Z    +0.000, E1    -9.693, E3 -170370.544}
SPL {X  -159.986, Y  +381.420, Z    +0.000, E1    -2.704, E3 -170371.109}
SPL {X  -159.990, Y  +384.527, Z    +0.000, E1    +0.013, E3 -170371.169}
SPL {X  -159.990, Y  +386.984, Z    +0.000, E1    +3.187, E3 -170371.221}
SPL {X  -159.990, Y  +390.572, Z    +0.000, E1    +9.243, E3 -170371.380}
SPL {X  -159.990, Y  +395.332, Z    +0.000, E1   +17.451, E3 -170371.794}
SPL {X  -159.990, Y  +403.857, Z    +0.000, E1   +31.979, E3 -170373.019}
SPL {X  -159.990, Y  +416.313, Z    +0.000, E1   +46.481, E3 -170376.012}
SPL {X  -159.990, Y  +425.447, Z    +0.000, E1   +52.896, E3 -170378.920}
SPL {X  -159.990, Y  +475.808, Z    +0.000, E1   +64.751, E3 -170400.458}
SPL {X  -159.990, Y  +586.159, Z    +0.000, E1   +66.648, E3 -170479.874}
SPL {X  -159.990, Y  +602.026, Z    +0.000, E1   +66.659, E3 -170494.391}
SPL {X  -159.990, Y  +615.972, Z    +0.000, E1   +66.639, E3 -170507.219}
SPL {X  -159.990, Y  +629.811, Z    +0.000, E1   +66.653, E3 -170519.871}
SPL {X  -159.990, Y  +646.024, Z    +0.000, E1   +66.650, E3 -170534.747}
SPL {X  -159.990, Y  +658.527, Z    +0.000, E1   +66.634, E3 -170546.229}
SPL {X  -159.990, Y  +671.049, Z    +0.000, E1   +66.648, E3 -170557.678}
SPL {X  -159.584, Y  +682.893, Z    +0.000, E1   +66.583, E3 -170568.976}
SPL {X  -158.332, Y  +694.472, Z    +0.000, E1   +66.450, E3 -170580.849}
SPL {X  -156.148, Y  +706.350, Z    +0.000, E1   +66.133, E3 -170594.061}
SPL {X  -154.052, Y  +714.685, Z    +0.000, E1   +65.842, E3 -170603.848}
SPL {X  -151.381, Y  +723.275, Z    +0.000, E1   +65.482, E3 -170614.395}
SPL {X  -147.622, Y  +733.180, Z    +0.000, E1   +64.943, E3 -170627.199}
SPL {X  -144.546, Y  +740.079, Z    +0.000, E1   +64.439, E3 -170636.527}
SPL {X  -141.166, Y  +746.792, Z    +0.000, E1   +63.950, E3 -170645.767}
SPL {X  -136.621, Y  +754.755, Z    +0.000, E1   +63.190, E3 -170657.163}
SPL {X  -133.172, Y  +760.168, Z    +0.000, E1   +62.565, E3 -170665.084}
SPL {X  -130.070, Y  +764.659, Z    +0.000, E1   +62.024, E3 -170671.680}
SPL {X  -103.420, Y  +793.570, Z    +0.000, E1   +51.337, E3 -170801.579}
ENDSPLINE

SPLINE
SPL {X  -141.359, Y  +746.429, Z    +0.000, E1   +41.207, E3 -170919.793}
SPL {X  -153.791, Y  +715.605, Z    +0.000, E1   +29.700, E3 -170934.562}
SPL {X  -157.923, Y  +697.131, Z    +0.000, E1   +19.758, E3 -170939.094}
SPL {X  -159.426, Y  +684.927, Z    +0.000, E1   +11.876, E3 -170940.823}
SPL {X  -159.972, Y  +673.894, Z    +0.000, E1    +3.783, E3 -170941.611}
SPL {X  -159.990, Y  +669.020, Z    +0.000, E1    -0.387, E3 -170941.715}
SPL {X  -159.990, Y  +664.217, Z    +0.000, E1    -7.944, E3 -170941.876}
SPL {X  -159.990, Y  +657.963, Z    +0.000, E1   -19.417, E3 -170942.372}
SPL {X  -159.990, Y  +649.570, Z    +0.000, E1   -33.681, E3 -170943.596}
SPL {X  -159.990, Y  +636.314, Z    +0.000, E1   -48.490, E3 -170946.900}
SPL {X  -159.990, Y  +588.081, Z    +0.000, E1   -63.406, E3 -170968.081}
SPL {X  -159.990, Y  +471.514, Z    +0.000, E1   -66.231, E3 -171051.589}
SPL {X  -159.990, Y  +458.012, Z    +0.000, E1   -66.224, E3 -171064.218}
SPL {X  -159.990, Y  +445.900, Z    +0.000, E1   -66.225, E3 -171075.532}
ENDSPLINE

SPLINE
SPL {X  -159.990, Y  +465.730, Z    +0.000, E1   -61.693, E3 -171089.356}
ENDSPLINE

SPLINE
SPL {X  -159.990, Y  +452.456, Z    +0.000, E1   -62.114, E3 -171101.284}
SPL {X  -159.990, Y  +436.367, Z    +0.000, E1   -62.893, E3 -171113.543}
SPL {X  -159.990, Y  +416.857, Z    +0.000, E1   -63.835, E3 -171127.282}
SPL {X  -159.990, Y  +397.192, Z    +0.000, E1   -64.622, E3 -171141.576}
SPL {X  -159.902, Y  +377.209, Z    +0.000, E1   -65.412, E3 -171155.140}
SPL {X  -158.342, Y  +359.598, Z    +0.000, E1   -66.150, E3 -171166.130}
SPL {X  -155.453, Y  +344.669, Z    +0.000, E1   -66.270, E3 -171178.972}
SPL {X  -152.827, Y  +335.165, Z    +0.000, E1   -65.880, E3 -171190.330}
SPL {X  -150.132, Y  +327.208, Z    +0.000, E1   -65.515, E3 -171200.223}
SPL {X  -147.311, Y  +320.081, Z    +0.000, E1   -65.083, E3 -171209.504}
SPL {X  -144.181, Y  +313.155, Z    +0.000, E1   -64.628, E3 -171218.765}
SPL {X  -141.300, Y  +307.460, Z    +0.000, E1   -64.150, E3 -171226.657}
SPL {X  -138.693, Y  +302.744, Z    +0.000, E1   -63.741, E3 -171233.271}
SPL {X  -135.031, Y  +296.690, Z    +0.000, E1   -63.147, E3 -171241.932}
SPL {X  -130.494, Y  +289.936, Z    +0.000, E1   -62.364, E3 -171251.770}
SPL {X  -102.192, Y  +259.400, Z    +0.000, E1   -52.167, E3 -171370.494}
ENDSPLINE

SPLINE
SPL {X  -140.725, Y  +306.386, Z    +0.000, E1   -41.058, E3 -171495.388}
SPL {X  -153.851, Y  +338.606, Z    +0.000, E1   -29.149, E3 -171512.006}
SPL {X  -158.264, Y  +359.064, Z    +0.000, E1   -18.155, E3 -171516.957}
SPL {X  -159.641, Y  +371.933, Z    +0.000, E1    -9.693, E3 -171518.692}
SPL {X  -159.986, Y  +381.420, Z    +0.000, E1    -2.704, E3 -171519.257}
SPL {X  -159.990, Y  +384.527, Z    +0.000, E1    +0.013, E3 -171519.318}
SPL {X  -159.990, Y  +385.909, Z    +0.000, E1    +1.800, E3 -171519.335}
SPL {X  -159.990, Y  +389.230, Z    +0.000, E1    +6.815, E3 -171519.459}
SPL {X  -159.990, Y  +395.332, Z    +0.000, E1   +17.451, E3 -171519.942}
SPL {X  -159.990, Y  +403.857, Z    +0.000, E1   +31.979, E3 -171521.167}
SPL {X  -159.990, Y  +417.858, Z    +0.000, E1   +47.695, E3 -171524.653}
SPL {X  -159.990, Y  +475.808, Z    +0.000, E1   +64.751, E3 -171548.606}
SPL {X  -159.990, Y  +586.159, Z    +0.000, E1   +66.648, E3 -171628.022}
SPL {X  -159.990, Y  +602.026, Z    +0.000, E1   +66.659, E3 -171642.539}
SPL {X  -159.990, Y  +620.525, Z    +0.000, E1   +66.669, E3 -171659.476}
SPL {X  -159.990, Y  +638.202, Z    +0.000, E1   +66.649, E3 -171675.726}
SPL {X  -159.990, Y  +654.774, Z    +0.000, E1   +66.658, E3 -171690.895}
SPL {X  -159.990, Y  +671.049, Z    +0.000, E1   +66.648, E3 -171705.826}
SPL {X  -159.230, Y  +687.071, Z    +0.000, E1   +66.569, E3 -171721.267}
SPL {X  -157.279, Y  +700.830, Z    +0.000, E1   +66.296, E3 -171735.957}
SPL {X  -154.589, Y  +712.719, Z    +0.000, E1   +65.941, E3 -171749.600}
SPL {X  -151.974, Y  +721.507, Z    +0.000, E1   +65.548, E3 -171760.353}
SPL {X  -149.510, Y  +728.452, Z    +0.000, E1   +65.197, E3 -171769.195}
SPL {X  -145.784, Y  +737.407, Z    +0.000, E1   +64.671, E3 -171780.986}
SPL {X  -142.587, Y  +744.066, Z    +0.000, E1   +64.133, E3 -171790.169}
SPL {X  -139.326, Y  +750.145, Z    +0.000, E1   +63.650, E3 -171798.662}
SPL {X  -135.791, Y  +756.103, Z    +0.000, E1   +63.018, E3 -171807.307}
SPL {X  -133.172, Y  +760.168, Z    +0.000, E1   +62.565, E3 -171813.232}
SPL {X  -130.070, Y  +764.659, Z    +0.000, E1   +62.024, E3 -171819.828}
SPL {X  -103.420, Y  +793.570, Z    +0.000, E1   +51.337, E3 -171949.727}
ENDSPLINE

SPLINE
SPL {X  -132.256, Y  +761.529, Z    +0.000, E1   +44.935, E3 -172055.817}
SPL {X  -148.790, Y  +730.309, Z    +0.000, E1   +35.907, E3 -172077.091}
SPL {X  -157.132, Y  +701.603, Z    +0.000, E1   +22.438, E3 -172086.352}
SPL {X  -159.426, Y  +684.927, Z    +0.000, E1   +11.876, E3 -172088.971}
SPL {X  -159.929, Y  +675.915, Z    +0.000, E1    +5.290, E3 -172089.681}
SPL {X  -159.990, Y  +669.794, Z    +0.000, E1    +0.371, E3 -172089.855}
SPL {X  -159.990, Y  +668.338, Z    +0.000, E1    -1.468, E3 -172089.871}
SPL {X  -159.990, Y  +665.597, Z    +0.000, E1    -5.793, E3 -172089.950}
SPL {X  -159.990, Y  +662.769, Z    +0.000, E1   -10.720, E3 -172090.101}
SPL {X  -159.990, Y  +658.787, Z    +0.000, E1   -17.995, E3 -172090.429}
SPL {X  -159.990, Y  +653.215, Z    +0.000, E1   -27.908, E3 -172091.121}
SPL {X  -159.990, Y  +646.194, Z    +0.000, E1   -38.517, E3 -172092.410}
SPL {X  -159.990, Y  +636.314, Z    +0.000, E1   -48.490, E3 -172095.048}
SPL {X  -159.990, Y  +588.081, Z    +0.000, E1   -63.406, E3 -172116.229}
SPL {X  -159.990, Y  +471.514, Z    +0.000, E1   -66.231, E3 -172199.737}
SPL {X  -159.990, Y  +458.012, Z    +0.000, E1   -66.224, E3 -172212.367}
SPL {X  -159.990, Y  +445.900, Z    +0.000, E1   -66.225, E3 -172223.680}
ENDSPLINE

SPLINE
SPL {X  -159.990, Y  +465.730, Z    +0.000, E1   -61.693, E3 -172237.504}
ENDSPLINE

SPLINE
SPL {X  -159.990, Y  +452.456, Z    +0.000, E1   -62.114, E3 -172249.432}
SPL {X  -159.990, Y  +436.367, Z    +0.000, E1   -62.893, E3 -172261.692}
SPL {X  -159.990, Y  +416.857, Z    +0.000, E1   -63.835, E3 -172275.431}
SPL {X  -159.990, Y  +397.192, Z    +0.000, E1   -64.622, E3 -172289.724}
SPL {X  -159.570, Y  +370.917, Z    +0.000, E1   -65.713, E3 -172307.081}
SPL {X  -156.693, Y  +350.188, Z    +0.000, E1   -66.345, E3 -172321.453}
SPL {X  -154.578, Y  +341.238, Z    +0.000, E1   -66.113, E3 -172331.211}
SPL {X  -151.958, Y  +332.444, Z    +0.000, E1   -65.791, E3 -172341.770}
SPL {X  -148.012, Y  +321.760, Z    +0.000, E1   -65.212, E3 -172355.404}
SPL {X  -144.181, Y  +313.155, Z    +0.000, E1   -64.628, E3 -172366.913}
SPL {X  -141.300, Y  +307.460, Z    +0.000, E1   -64.150, E3 -172374.805}
SPL {X  -138.693, Y  +302.744, Z    +0.000, E1   -63.741, E3 -172381.419}
SPL {X  -135.977, Y  +298.197, Z    +0.000, E1   -63.280, E3 -172387.939}
SPL {X  -132.828, Y  +293.318, Z    +0.000, E1   -62.759, E3 -172394.992}
SPL {X  -129.451, Y  +288.482, Z    +0.000, E1   -62.137, E3 -172402.096}
SPL {X  -102.192, Y  +259.400, Z    +0.000, E1   -52.167, E3 -172518.643}
ENDSPLINE

SPLINE
SPL {X  -140.725, Y  +306.386, Z    +0.000, E1   -41.058, E3 -172643.537}
SPL {X  -153.851, Y  +338.606, Z    +0.000, E1   -29.149, E3 -172660.154}
SPL {X  -157.523, Y  +354.512, Z    +0.000, E1   -20.811, E3 -172664.280}
SPL {X  -159.458, Y  +369.460, Z    +0.000, E1   -11.469, E3 -172666.569}
SPL {X  -159.986, Y  +381.420, Z    +0.000, E1    -2.704, E3 -172667.405}
SPL {X  -159.990, Y  +384.527, Z    +0.000, E1    +0.013, E3 -172667.466}
SPL {X  -159.990, Y  +385.909, Z    +0.000, E1    +1.800, E3 -172667.483}
SPL {X  -159.990, Y  +389.230, Z    +0.000, E1    +6.815, E3 -172667.608}
SPL {X  -159.990, Y  +395.332, Z    +0.000, E1   +17.451, E3 -172668.090}
SPL {X  -159.990, Y  +403.857, Z    +0.000, E1   +31.979, E3 -172669.316}
SPL {X  -159.990, Y  +417.858, Z    +0.000, E1   +47.695, E3 -172672.801}
SPL {X  -159.990, Y  +475.808, Z    +0.000, E1   +64.751, E3 -172696.754}
SPL {X  -159.990, Y  +590.266, Z    +0.000, E1   +66.680, E3 -172779.872}
SPL {X  -159.990, Y  +611.678, Z    +0.000, E1   +66.672, E3 -172799.511}
SPL {X  -159.990, Y  +625.813, Z    +0.000, E1   +66.632, E3 -172812.543}
SPL {X  -159.990, Y  +638.202, Z    +0.000, E1   +66.649, E3 -172823.874}
SPL {X  -159.990, Y  +654.774, Z    +0.000, E1   +66.658, E3 -172839.043}
SPL {X  -159.990, Y  +671.049, Z    +0.000, E1   +66.648, E3 -172853.974}
SPL {X  -159.584, Y  +682.893, Z    +0.000, E1   +66.583, E3 -172865.272}
SPL {X  -158.332, Y  +694.472, Z    +0.000, E1   +66.450, E3 -172877.145}
SPL {X  -156.148, Y  +706.350, Z    +0.000, E1   +66.133, E3 -172890.357}
SPL {X  -154.052, Y  +714.685, Z    +0.000, E1   +65.842, E3 -172900.144}
SPL {X  -151.381, Y  +723.275, Z    +0.000, E1   +65.482, E3 -172910.691}
SPL {X  -147.622, Y  +733.180, Z    +0.000, E1   +64.943, E3 -172923.495}
SPL {X  -144.546, Y  +740.079, Z    +0.000, E1   +64.439, E3 -172932.823}
SPL {X  -142.587, Y  +744.066, Z    +0.000, E1   +64.133, E3 -172938.317}
SPL {X  -139.326, Y  +750.145, Z    +0.000, E1   +63.650, E3 -172946.810}
SPL {X  -135.791, Y  +756.103, Z    +0.000, E1   +63.018, E3 -172955.456}
SPL {X  -133.172, Y  +760.168, Z    +0.000, E1   +62.565, E3 -172961.380}
SPL {X  -130.070, Y  +764.659, Z    +0.000, E1   +62.024, E3 -172967.976}
SPL {X  -103.420, Y  +793.570, Z    +0.000, E1   +51.337, E3 -173097.876}
ENDSPLINE

SPLINE
SPL {X  -132.256, Y  +761.529, Z    +0.000, E1   +44.935, E3 -173203.965}
SPL {X  -148.790, Y  +730.309, Z    +0.000, E1   +35.907, E3 -173225.239}
SPL {X  -157.132, Y  +701.603, Z    +0.000, E1   +22.438, E3 -173234.500}
SPL {X  -159.426, Y  +684.927, Z    +0.000, E1   +11.876, E3 -173237.119}
SPL {X  -159.972, Y  +673.894, Z    +0.000, E1    +3.783, E3 -173237.907}
SPL {X  -159.990, Y  +669.020, Z    +0.000, E1    -0.387, E3 -173238.012}
SPL {X  -159.990, Y  +664.217, Z    +0.000, E1    -7.944, E3 -173238.172}
SPL {X  -159.990, Y  +657.963, Z    +0.000, E1   -19.417, E3 -173238.669}
SPL {X  -159.990, Y  +649.570, Z    +0.000, E1   -33.681, E3 -173239.893}
SPL {X  -159.990, Y  +636.314, Z    +0.000, E1   -48.490, E3 -173243.196}
SPL {X  -159.990, Y  +588.081, Z    +0.000, E1   -63.406, E3 -173264.377}
SPL {X  -159.990, Y  +471.514, Z    +0.000, E1   -66.231, E3 -173347.885}
SPL {X  -159.990, Y  +458.012, Z    +0.000, E1   -66.224, E3 -173360.515}
SPL {X  -159.990, Y  +445.900, Z    +0.000, E1   -66.225, E3 -173371.828}
ENDSPLINE

SPLINE
SPL {X  -159.990, Y  +468.953, Z    +0.000, E1   -61.697, E3 -173381.786}
ENDSPLINE

SPLINE
SPL {X  -159.990, Y  +457.098, Z    +0.000, E1   -61.912, E3 -173393.883}
SPL {X  -159.990, Y  +442.075, Z    +0.000, E1   -62.596, E3 -173405.658}
SPL {X  -159.990, Y  +430.868, Z    +0.000, E1   -63.135, E3 -173413.912}
SPL {X  -159.990, Y  +416.857, Z    +0.000, E1   -63.835, E3 -173423.579}
SPL {X  -159.990, Y  +397.192, Z    +0.000, E1   -64.622, E3 -173437.872}
SPL {X  -159.570, Y  +370.917, Z    +0.000, E1   -65.713, E3 -173455.229}
SPL {X  -156.693, Y  +350.188, Z    +0.000, E1   -66.345, E3 -173469.601}
SPL {X  -153.533, Y  +337.508, Z    +0.000, E1   -66.008, E3 -173483.733}
SPL {X  -150.132, Y  +327.208, Z    +0.000, E1   -65.515, E3 -173496.519}
SPL {X  -146.325, Y  +317.802, Z    +0.000, E1   -64.967, E3 -173508.774}
SPL {X  -142.205, Y  +309.188, Z    +0.000, E1   -64.322, E3 -173520.510}
SPL {X  -138.693, Y  +302.744, Z    +0.000, E1   -63.741, E3 -173529.567}
SPL {X  -135.031, Y  +296.690, Z    +0.000, E1   -63.147, E3 -173538.228}
SPL {X  -130.494, Y  +289.936, Z    +0.000, E1   -62.364, E3 -173548.066}
SPL {X  -102.192, Y  +259.400, Z    +0.000, E1   -52.167, E3 -173666.791}
ENDSPLINE

SPLINE
SPL {X  -140.725, Y  +306.386, Z    +0.000, E1   -41.058, E3 -173791.685}
SPL {X  -153.851, Y  +338.606, Z    +0.000, E1   -29.149, E3 -173808.302}
SPL {X  -157.523, Y  +354.512, Z    +0.000, E1   -20.811, E3 -173812.428}
SPL {X  -159.458, Y  +369.460, Z    +0.000, E1   -11.469, E3 -173814.718}
SPL {X  -159.986, Y  +381.420, Z    +0.000, E1    -2.704, E3 -173815.553}
SPL {X  -159.990, Y  +385.016, Z    +0.000, E1    +0.442, E3 -173815.620}
SPL {X  -159.990, Y  +389.230, Z    +0.000, E1    +6.815, E3 -173815.756}
SPL {X  -159.990, Y  +393.768, Z    +0.000, E1   +14.836, E3 -173816.074}
SPL {X  -159.990, Y  +397.827, Z    +0.000, E1   +22.184, E3 -173816.500}
SPL {X  -159.990, Y  +403.857, Z    +0.000, E1   +31.979, E3 -173817.464}
SPL {X  -159.990, Y  +417.858, Z    +0.000, E1   +47.695, E3 -173820.949}
SPL {X  -159.990, Y  +475.808, Z    +0.000, E1   +64.751, E3 -173844.902}
SPL {X  -159.990, Y  +590.266, Z    +0.000, E1   +66.680, E3 -173928.020}
SPL {X  -159.990, Y  +605.903, Z    +0.000, E1   +66.635, E3 -173942.439}
SPL {X  -159.990, Y  +620.525, Z    +0.000, E1   +66.669, E3 -173955.773}
SPL {X  -159.990, Y  +638.202, Z    +0.000, E1   +66.649, E3 -173972.022}
SPL {X  -159.990, Y  +649.814, Z    +0.000, E1   +66.629, E3 -173982.710}
SPL {X  -159.990, Y  +658.527, Z    +0.000, E1   +66.634, E3 -173990.673}
SPL {X  -159.990, Y  +671.049, Z    +0.000, E1   +66.648, E3 -174002.122}
SPL {X  -159.584, Y  +682.893, Z    +0.000, E1   +66.583, E3 -174013.420}
SPL {X  -158.332, Y  +694.472, Z    +0.000, E1   +66.450, E3 -174025.294}
SPL {X  -156.148, Y  +706.350, Z    +0.000, E1   +66.133, E3 -174038.505}
SPL {X  -154.052, Y  +714.685, Z    +0.000, E1   +65.842, E3 -174048.292}
SPL {X  -151.974, Y  +721.507, Z    +0.000, E1   +65.548, E3 -174056.649}
SPL {X  -149.510, Y  +728.452, Z    +0.000, E1   +65.197, E3 -174065.492}
SPL {X  -146.809, Y  +735.092, Z    +0.000, E1   +64.789, E3 -174074.239}
SPL {X  -143.550, Y  +742.141, Z    +0.000, E1   +64.312, E3 -174083.757}
SPL {X  -140.309, Y  +748.378, Z    +0.000, E1   +63.779, E3 -174092.490}
SPL {X  -136.621, Y  +754.755, Z    +0.000, E1   +63.190, E3 -174101.607}
SPL {X  -133.172, Y  +760.168, Z    +0.000, E1   +62.565, E3 -174109.528}
SPL {X  -130.070, Y  +764.659, Z    +0.000, E1   +62.024, E3 -174116.124}
SPL {X  -103.420, Y  +793.570, Z    +0.000, E1   +51.337, E3 -174246.024}
ENDSPLINE

SPLINE
SPL {X  -132.256, Y  +761.529, Z    +0.000, E1   +44.935, E3 -174352.113}
SPL {X  -148.790, Y  +730.309, Z    +0.000, E1   +35.907, E3 -174373.387}
SPL {X  -157.132, Y  +701.603, Z    +0.000, E1   +22.438, E3 -174382.648}
SPL {X  -159.426, Y  +684.927, Z    +0.000, E1   +11.876, E3 -174385.267}
SPL {X  -159.929, Y  +675.915, Z    +0.000, E1    +5.290, E3 -174385.977}
SPL {X  -159.990, Y  +669.794, Z    +0.000, E1    +0.371, E3 -174386.151}
SPL {X  -159.990, Y  +668.338, Z    +0.000, E1    -1.468, E3 -174386.168}
SPL {X  -159.990, Y  +664.217, Z    +0.000, E1    -7.944, E3 -174386.320}
SPL {X  -159.990, Y  +658.787, Z    +0.000, E1   -17.995, E3 -174386.725}
SPL {X  -159.990, Y  +653.215, Z    +0.000, E1   -27.908, E3 -174387.417}
SPL {X  -159.990, Y  +646.194, Z    +0.000, E1   -38.517, E3 -174388.706}
SPL {X  -159.990, Y  +636.314, Z    +0.000, E1   -48.490, E3 -174391.344}
SPL {X  -159.990, Y  +588.081, Z    +0.000, E1   -63.406, E3 -174412.525}
SPL {X  -159.990, Y  +471.514, Z    +0.000, E1   -66.231, E3 -174496.033}
SPL {X  -159.990, Y  +458.012, Z    +0.000, E1   -66.224, E3 -174508.663}
SPL {X  -159.990, Y  +445.900, Z    +0.000, E1   -66.225, E3 -174519.976}
ENDSPLINE

SPLINE
SPL {X  -159.990, Y  +465.730, Z    +0.000, E1   -61.693, E3 -174533.801}
ENDSPLINE

SPLINE
SPL {X  -159.990, Y  +452.456, Z    +0.000, E1   -62.114, E3 -174545.728}
SPL {X  -159.990, Y  +436.367, Z    +0.000, E1   -62.893, E3 -174557.988}
SPL {X  -159.990, Y  +416.857, Z    +0.000, E1   -63.835, E3 -174571.727}
SPL {X  -159.990, Y  +397.192, Z    +0.000, E1   -64.622, E3 -174586.020}
SPL {X  -159.902, Y  +377.209, Z    +0.000, E1   -65.412, E3 -174599.584}
SPL {X  -158.342, Y  +359.598, Z    +0.000, E1   -66.150, E3 -174610.575}
SPL {X  -155.453, Y  +344.669, Z    +0.000, E1   -66.270, E3 -174623.417}
SPL {X  -152.827, Y  +335.165, Z    +0.000, E1   -65.880, E3 -174634.774}
SPL {X  -150.132, Y  +327.208, Z    +0.000, E1   -65.515, E3 -174644.667}
SPL {X  -147.311, Y  +320.081, Z    +0.000, E1   -65.083, E3 -174653.948}
SPL {X  -144.181, Y  +313.155, Z    +0.000, E1   -64.628, E3 -174663.209}
SPL {X  -141.300, Y  +307.460, Z    +0.000, E1   -64.150, E3 -174671.101}
SPL {X  -138.693, Y  +302.744, Z    +0.000, E1   -63.741, E3 -174677.715}
SPL {X  -135.977, Y  +298.197, Z    +0.000, E1   -63.280, E3 -174684.235}
SPL {X  -132.828, Y  +293.318, Z    +0.000, E1   -62.759, E3 -174691.288}
SPL {X  -129.451, Y  +288.482, Z    +0.000, E1   -62.137, E3 -174698.392}
SPL {X  -102.192, Y  +259.400, Z    +0.000, E1   -52.167, E3 -174814.939}
ENDSPLINE

SPLINE
SPL {X  -140.725, Y  +306.386, Z    +0.000, E1   -41.058, E3 -174939.833}
SPL {X  -153.851, Y  +338.606, Z    +0.000, E1   -29.149, E3 -174956.450}
SPL {X  -158.264, Y  +359.064, Z    +0.000, E1   -18.155, E3 -174961.401}
SPL {X  -159.641, Y  +371.933, Z    +0.000, E1    -9.693, E3 -174963.136}
SPL {X  -159.986, Y  +381.420, Z    +0.000, E1    -2.704, E3 -174963.701}
SPL {X  -159.990, Y  +384.527, Z    +0.000, E1    +0.013, E3 -174963.762}
SPL {X  -159.990, Y  +385.909, Z    +0.000, E1    +1.800, E3 -174963.779}
SPL {X  -159.990, Y  +389.230, Z    +0.000, E1    +6.815, E3 -174963.904}
SPL {X  -159.990, Y  +395.332, Z    +0.000, E1   +17.451, E3 -174964.387}
SPL {X  -159.990, Y  +403.857, Z    +0.000, E1   +31.979, E3 -174965.612}
SPL {X  -159.990, Y  +417.858, Z    +0.000, E1   +47.695, E3 -174969.097}
SPL {X  -159.990, Y  +475.808, Z    +0.000, E1   +64.751, E3 -174993.051}
SPL {X  -159.990, Y  +586.159, Z    +0.000, E1   +66.648, E3 -175072.467}
SPL {X  -159.990, Y  +602.026, Z    +0.000, E1   +66.659, E3 -175086.983}
SPL {X  -159.990, Y  +620.525, Z    +0.000, E1   +66.669, E3 -175103.921}
SPL {X  -159.990, Y  +638.202, Z    +0.000, E1   +66.649, E3 -175120.171}
SPL {X  -159.990, Y  +654.774, Z    +0.000, E1   +66.658, E3 -175135.340}
SPL {X  -159.990, Y  +671.049, Z    +0.000, E1   +66.648, E3 -175150.270}
SPL {X  -159.230, Y  +687.071, Z    +0.000, E1   +66.569, E3 -175165.712}
SPL {X  -157.279, Y  +700.830, Z    +0.000, E1   +66.296, E3 -175180.402}
SPL {X  -154.589, Y  +712.719, Z    +0.000, E1   +65.941, E3 -175194.045}
SPL {X  -151.381, Y  +723.275, Z    +0.000, E1   +65.482, E3 -175206.988}
SPL {X  -147.622, Y  +733.180, Z    +0.000, E1   +64.943, E3 -175219.791}
SPL {X  -143.550, Y  +742.141, Z    +0.000, E1   +64.312, E3 -175231.905}
SPL {X  -139.326, Y  +750.145, Z    +0.000, E1   +63.650, E3 -175243.107}
SPL {X  -135.791, Y  +756.103, Z    +0.000, E1   +63.018, E3 -175251.752}
SPL {X  -133.172, Y  +760.168, Z    +0.000, E1   +62.565, E3 -175257.677}
SPL {X  -130.070, Y  +764.659, Z    +0.000, E1   +62.024, E3 -175264.272}
SPL {X  -103.420, Y  +793.570, Z    +0.000, E1   +51.337, E3 -175394.172}
ENDSPLINE

SPLINE
SPL {X  -141.359, Y  +746.429, Z    +0.000, E1   +41.207, E3 -175512.386}
SPL {X  -153.791, Y  +715.605, Z    +0.000, E1   +29.700, E3 -175527.155}
SPL {X  -157.923, Y  +697.131, Z    +0.000, E1   +19.758, E3 -175531.686}
SPL {X  -159.426, Y  +684.927, Z    +0.000, E1   +11.876, E3 -175533.415}
SPL {X  -159.972, Y  +673.894, Z    +0.000, E1    +3.783, E3 -175534.203}
SPL {X  -159.990, Y  +669.561, Z    +0.000, E1    +0.077, E3 -175534.302}
SPL {X  -159.990, Y  +668.338, Z    +0.000, E1    -1.468, E3 -175534.316}
SPL {X  -159.990, Y  +664.217, Z    +0.000, E1    -7.944, E3 -175534.468}
SPL {X  -159.990, Y  +658.787, Z    +0.000, E1   -17.995, E3 -175534.873}
SPL {X  -159.990, Y  +653.215, Z    +0.000, E1   -27.908, E3 -175535.565}
SPL {X  -159.990, Y  +646.194, Z    +0.000, E1   -38.517, E3 -175536.854}
SPL {X  -159.990, Y  +636.314, Z    +0.000, E1   -48.490, E3 -175539.492}
SPL {X  -159.990, Y  +588.081, Z    +0.000, E1   -63.406, E3 -175560.674}
SPL {X  -159.990, Y  +471.514, Z    +0.000, E1   -66.231, E3 -175644.182}
SPL {X  -159.990, Y  +458.012, Z    +0.000, E1   -66.224, E3 -175656.811}
SPL {X  -159.990, Y  +445.900, Z    +0.000, E1   -66.225, E3 -175668.124}
ENDSPLINE

SPLINE
SPL {X  -159.990, Y  +465.730, Z    +0.000, E1   -61.693, E3 -175681.949}
ENDSPLINE

SPLINE
SPL {X  -159.990, Y  +446.910, Z    +0.000, E1   -62.394, E3 -175698.168}
SPL {X  -159.990, Y  +430.868, Z    +0.000, E1   -63.135, E3 -175710.208}
SPL {X  -159.990, Y  +416.857, Z    +0.000, E1   -63.835, E3 -175719.875}
SPL {X  -159.990, Y  +397.192, Z    +0.000, E1   -64.622, E3 -175734.168}
SPL {X  -159.570, Y  +370.917, Z    +0.000, E1   -65.713, E3 -175751.525}
SPL {X  -156.693, Y  +350.188, Z    +0.000, E1   -66.345, E3 -175765.897}
SPL {X  -153.533, Y  +337.508, Z    +0.000, E1   -66.008, E3 -175780.029}
SPL {X  -150.132, Y  +327.208, Z    +0.000, E1   -65.515, E3 -175792.815}
SPL {X  -146.325, Y  +317.802, Z    +0.000, E1   -64.967, E3 -175805.070}
SPL {X  -142.205, Y  +309.188, Z    +0.000, E1   -64.322, E3 -175816.806}
SPL {X  -138.693, Y  +302.744, Z    +0.000, E1   -63.741, E3 -175825.863}
SPL {X  -135.977, Y  +298.197, Z    +0.000, E1   -63.280, E3 -175832.383}
SPL {X  -132.828, Y  +293.318, Z    +0.000, E1   -62.759, E3 -175839.436}
SPL {X  -129.451, Y  +288.482, Z    +0.000, E1   -62.137, E3 -175846.540}
SPL {X  -102.192, Y  +259.400, Z    +0.000, E1   -52.167, E3 -175963.087}
ENDSPLINE

SPLINE
SPL {X  -140.725, Y  +306.386, Z    +0.000, E1   -41.058, E3 -176087.981}
SPL {X  -153.851, Y  +338.606, Z    +0.000, E1   -29.149, E3 -176104.598}
SPL {X  -158.264, Y  +359.064, Z    +0.000, E1   -18.155, E3 -176109.549}
SPL {X  -159.641, Y  +371.933, Z    +0.000, E1    -9.693, E3 -176111.284}
SPL {X  -159.986, Y  +381.420, Z    +0.000, E1    -2.704, E3 -176111.850}
SPL {X  -159.990, Y  +384.527, Z    +0.000, E1    +0.013, E3 -176111.910}
SPL {X  -159.990, Y  +386.984, Z    +0.000, E1    +3.187, E3 -176111.962}
SPL {X  -159.990, Y  +390.572, Z    +0.000, E1    +9.243, E3 -176112.121}
SPL {X  -159.990, Y  +395.332, Z    +0.000, E1   +17.451, E3 -176112.535}
SPL {X  -159.990, Y  +403.857, Z    +0.000, E1   +31.979, E3 -176113.760}
SPL {X  -159.990, Y  +416.313, Z    +0.000, E1   +46.481, E3 -176116.752}
SPL {X  -159.990, Y  +425.447, Z    +0.000, E1   +52.896, E3 -176119.661}
SPL {X  -159.990, Y  +475.808, Z    +0.000, E1   +64.751, E3 -176141.199}
SPL {X  -159.990, Y  +590.266, Z    +0.000, E1   +66.680, E3 -176224.316}
SPL {X  -159.990, Y  +611.678, Z    +0.000, E1   +66.672, E3 -176243.956}
SPL {X  -159.990, Y  +629.811, Z    +0.000, E1   +66.653, E3 -176260.612}
SPL {X  -159.990, Y  +646.024, Z    +0.000, E1   +66.650, E3 -176275.488}
SPL {X  -159.990, Y  +658.527, Z    +0.000, E1   +66.634, E3 -176286.970}
SPL {X  -159.990, Y  +671.049, Z    +0.000, E1   +66.648, E3 -176298.419}
SPL {X  -159.584, Y  +682.893, Z    +0.000, E1   +66.583, E3 -176309.716}
SPL {X  -158.332, Y  +694.472, Z    +0.000, E1   +66.450, E3 -176321.590}
SPL {X  -156.148, Y  +706.350, Z    +0.000, E1   +66.133, E3 -176334.801}
SPL {X  -154.052, Y  +714.685, Z    +0.000, E1   +65.842, E3 -176344.589}
SPL {X  -151.974, Y  +721.507, Z    +0.000, E1   +65.548, E3 -176352.945}
SPL {X  -149.510, Y  +728.452, Z    +0.000, E1   +65.197, E3 -176361.788}
SPL {X  -145.784, Y  +737.407, Z    +0.000, E1   +64.671, E3 -176373.579}
SPL {X  -142.587, Y  +744.066, Z    +0.000, E1   +64.133, E3 -176382.762}
SPL {X  -139.326, Y  +750.145, Z    +0.000, E1   +63.650, E3 -176391.255}
SPL {X  -135.791, Y  +756.103, Z    +0.000, E1   +63.018, E3 -176399.900}
SPL {X  -133.172, Y  +760.168, Z    +0.000, E1   +62.565, E3 -176405.825}
SPL {X  -130.070, Y  +764.659, Z    +0.000, E1   +62.024, E3 -176412.420}
SPL {X  -103.420, Y  +793.570, Z    +0.000, E1   +51.337, E3 -176542.320}
ENDSPLINE

SPLINE
SPL {X  -132.256, Y  +761.529, Z    +0.000, E1   +44.935, E3 -176648.410}
SPL {X  -148.790, Y  +730.309, Z    +0.000, E1   +35.907, E3 -176669.683}
SPL {X  -157.132, Y  +701.603, Z    +0.000, E1   +22.438, E3 -176678.944}
SPL {X  -159.426, Y  +684.927, Z    +0.000, E1   +11.876, E3 -176681.563}
SPL {X  -159.929, Y  +675.915, Z    +0.000, E1    +5.290, E3 -176682.274}
SPL {X  -159.990, Y  +669.794, Z    +0.000, E1    +0.371, E3 -176682.447}
SPL {X  -159.990, Y  +668.338, Z    +0.000, E1    -1.468, E3 -176682.464}
SPL {X  -159.990, Y  +665.597, Z    +0.000, E1    -5.793, E3 -176682.543}
SPL {X  -159.990, Y  +662.769, Z    +0.000, E1   -10.720, E3 -176682.694}
SPL {X  -159.990, Y  +658.787, Z    +0.000, E1   -17.995, E3 -176683.022}
SPL {X  -159.990, Y  +653.215, Z    +0.000, E1   -27.908, E3 -176683.714}
SPL {X  -159.990, Y  +646.194, Z    +0.000, E1   -38.517, E3 -176685.002}
SPL {X  -159.990, Y  +636.314, Z    +0.000, E1   -48.490, E3 -176687.640}
SPL {X  -159.990, Y  +588.081, Z    +0.000, E1   -63.406, E3 -176708.822}
SPL {X  -159.990, Y  +471.514, Z    +0.000, E1   -66.231, E3 -176792.330}
SPL {X  -159.990, Y  +458.012, Z    +0.000, E1   -66.224, E3 -176804.959}
SPL {X  -159.990, Y  +445.900, Z    +0.000, E1   -66.225, E3 -176816.272}
ENDSPLINE

SPLINE
SPL {X  -159.990, Y  +468.953, Z    +0.000, E1   -61.697, E3 -176826.231}
ENDSPLINE

SPLINE
SPL {X  -159.990, Y  +457.098, Z    +0.000, E1   -61.912, E3 -176838.327}
SPL {X  -159.990, Y  +442.075, Z    +0.000, E1   -62.596, E3 -176850.103}
SPL {X  -159.990, Y  +430.868, Z    +0.000, E1   -63.135, E3 -176858.356}
SPL {X  -159.990, Y  +416.857, Z    +0.000, E1   -63.835, E3 -176868.023}
SPL {X  -159.990, Y  +402.942, Z    +0.000, E1   -64.377, E3 -176878.252}
SPL {X  -159.990, Y  +382.745, Z    +0.000, E1   -65.209, E3 -176892.166}
SPL {X  -158.929, Y  +364.101, Z    +0.000, E1   -65.981, E3 -176903.921}
SPL {X  -156.693, Y  +350.188, Z    +0.000, E1   -66.345, E3 -176914.045}
SPL {X  -154.578, Y  +341.238, Z    +0.000, E1   -66.113, E3 -176923.803}
SPL {X  -151.958, Y  +332.444, Z    +0.000, E1   -65.791, E3 -176934.363}
SPL {X  -148.012, Y  +321.760, Z    +0.000, E1   -65.212, E3 -176947.996}
SPL {X  -145.172, Y  +315.256, Z    +0.000, E1   -64.753, E3 -176956.701}
SPL {X  -142.205, Y  +309.188, Z    +0.000, E1   -64.322, E3 -176964.954}
SPL {X  -138.693, Y  +302.744, Z    +0.000, E1   -63.741, E3 -176974.011}
SPL {X  -135.977, Y  +298.197, Z    +0.000, E1   -63.280, E3 -176980.531}
SPL {X  -132.828, Y  +293.318, Z    +0.000, E1   -62.759, E3 -176987.585}
SPL {X  -129.451, Y  +288.482, Z    +0.000, E1   -62.137, E3 -176994.688}
SPL {X  -102.192, Y  +259.400, Z    +0.000, E1   -52.167, E3 -177111.235}
ENDSPLINE

SPLINE
SPL {X  -140.725, Y  +306.386, Z    +0.000, E1   -41.058, E3 -177236.129}
SPL {X  -153.851, Y  +338.606, Z    +0.000, E1   -29.149, E3 -177252.746}
SPL {X  -158.264, Y  +359.064, Z    +0.000, E1   -18.155, E3 -177257.697}
SPL {X  -159.641, Y  +371.933, Z    +0.000, E1    -9.693, E3 -177259.433}
SPL {X  -159.986, Y  +381.420, Z    +0.000, E1    -2.704, E3 -177259.998}
SPL {X  -159.990, Y  +384.527, Z    +0.000, E1    +0.013, E3 -177260.058}
SPL {X  -159.990, Y  +385.909, Z    +0.000, E1    +1.800, E3 -177260.076}
SPL {X  -159.990, Y  +389.230, Z    +0.000, E1    +6.815, E3 -177260.200}
SPL {X  -159.990, Y  +395.332, Z    +0.000, E1   +17.451, E3 -177260.683}
SPL {X  -159.990, Y  +403.857, Z    +0.000, E1   +31.979, E3 -177261.908}
SPL {X  -159.990, Y  +417.858, Z    +0.000, E1   +47.695, E3 -177265.393}
SPL {X  -159.990, Y  +475.808, Z    +0.000, E1   +64.751, E3 -177289.347}
SPL {X  -159.990, Y  +590.266, Z    +0.000, E1   +66.680, E3 -177372.464}
SPL {X  -159.990, Y  +605.903, Z    +0.000, E1   +66.635, E3 -177386.883}
SPL {X  -159.990, Y  +620.525, Z    +0.000, E1   +66.669, E3 -177400.217}
SPL {X  -159.990, Y  +638.202, Z    +0.000, E1   +66.649, E3 -177416.467}
SPL {X  -159.990, Y  +654.774, Z    +0.000, E1   +66.658, E3 -177431.636}
SPL {X  -159.990, Y  +671.049, Z    +0.000, E1   +66.648, E3 -177446.567}
SPL {X  -159.584, Y  +682.893, Z    +0.000, E1   +66.583, E3 -177457.864}
SPL {X  -158.845, Y  +690.607, Z    +0.000, E1   +66.486, E3 -177465.717}
SPL {X  -157.279, Y  +700.830, Z    +0.000, E1   +66.296, E3 -177476.698}
SPL {X  -154.589, Y  +712.719, Z    +0.000, E1   +65.941, E3 -177490.341}
SPL {X  -151.974, Y  +721.507, Z    +0.000, E1   +65.548, E3 -177501.093}
SPL {X  -149.510, Y  +728.452, Z    +0.000, E1   +65.197, E3 -177509.936}
SPL {X  -146.809, Y  +735.092, Z    +0.000, E1   +64.789, E3 -177518.683}
SPL {X  -143.550, Y  +742.141, Z    +0.000, E1   +64.312, E3 -177528.202}
SPL {X  -140.309, Y  +748.378, Z    +0.000, E1   +63.779, E3 -177536.935}
SPL {X  -136.621, Y  +754.755, Z    +0.000, E1   +63.190, E3 -177546.052}
SPL {X  -133.172, Y  +760.168, Z    +0.000, E1   +62.565, E3 -177553.973}
SPL {X  -130.070, Y  +764.659, Z    +0.000, E1   +62.024, E3 -177560.568}
SPL {X  -103.420, Y  +793.570, Z    +0.000, E1   +51.337, E3 -177690.468}
ENDSPLINE

SPLINE
SPL {X  -141.359, Y  +746.429, Z    +0.000, E1   +41.207, E3 -177808.682}
SPL {X  -153.791, Y  +715.605, Z    +0.000, E1   +29.700, E3 -177823.451}
SPL {X  -157.923, Y  +697.131, Z    +0.000, E1   +19.758, E3 -177827.983}
SPL {X  -159.426, Y  +684.927, Z    +0.000, E1   +11.876, E3 -177829.711}
SPL {X  -159.929, Y  +675.915, Z    +0.000, E1    +5.290, E3 -177830.422}
SPL {X  -159.990, Y  +669.794, Z    +0.000, E1    +0.371, E3 -177830.595}
SPL {X  -159.990, Y  +668.338, Z    +0.000, E1    -1.468, E3 -177830.612}
SPL {X  -159.990, Y  +664.217, Z    +0.000, E1    -7.944, E3 -177830.764}
SPL {X  -159.990, Y  +657.963, Z    +0.000, E1   -19.417, E3 -177831.261}
SPL {X  -159.990, Y  +649.570, Z    +0.000, E1   -33.681, E3 -177832.485}
SPL {X  -159.990, Y  +636.314, Z    +0.000, E1   -48.490, E3 -177835.788}
SPL {X  -159.990, Y  +588.081, Z    +0.000, E1   -63.406, E3 -177856.970}
SPL {X  -159.990, Y  +471.514, Z    +0.000, E1   -66.231, E3 -177940.478}
SPL {X  -159.990, Y  +458.012, Z    +0.000, E1   -66.224, E3 -177953.107}
SPL {X  -159.990, Y  +445.900, Z    +0.000, E1   -66.225, E3 -177964.421}
ENDSPLINE

SPLINE
SPL {X  -159.990, Y  +465.730, Z    +0.000, E1   -61.693, E3 -177978.245}
ENDSPLINE

SPLINE
SPL {X  -159.990, Y  +446.910, Z    +0.000, E1   -62.394, E3 -177994.465}
SPL {X  -159.990, Y  +430.868, Z    +0.000, E1   -63.135, E3 -178006.504}
SPL {X  -159.990, Y  +416.857, Z    +0.000, E1   -63.835, E3 -178016.171}
SPL {X  -159.990, Y  +402.942, Z    +0.000, E1   -64.377, E3 -178026.400}
SPL {X  -159.990, Y  +382.745, Z    +0.000, E1   -65.209, E3 -178040.314}
SPL {X  -158.342, Y  +359.598, Z    +0.000, E1   -66.150, E3 -178055.019}
SPL {X  -155.453, Y  +344.669, Z    +0.000, E1   -66.270, E3 -178067.861}
SPL {X  -151.958, Y  +332.444, Z    +0.000, E1   -65.791, E3 -178082.511}
SPL {X  -148.012, Y  +321.760, Z    +0.000, E1   -65.212, E3 -178096.144}
SPL {X  -144.181, Y  +313.155, Z    +0.000, E1   -64.628, E3 -178107.654}
SPL {X  -141.300, Y  +307.460, Z    +0.000, E1   -64.150, E3 -178115.546}
SPL {X  -138.693, Y  +302.744, Z    +0.000, E1   -63.741, E3 -178122.159}
SPL {X  -135.031, Y  +296.690, Z    +0.000, E1   -63.147, E3 -178130.821}
SPL {X  -130.494, Y  +289.936, Z    +0.000, E1   -62.364, E3 -178140.659}
SPL {X  -102.192, Y  +259.400, Z    +0.000, E1   -52.167, E3 -178259.383}
ENDSPLINE

SPLINE
SPL {X  -140.725, Y  +306.386, Z    +0.000, E1   -41.058, E3 -178384.277}
SPL {X  -153.851, Y  +338.606, Z    +0.000, E1   -29.149, E3 -178400.895}
SPL {X  -158.264, Y  +359.064, Z    +0.000, E1   -18.155, E3 -178405.846}
SPL {X  -159.641, Y  +371.933, Z    +0.000, E1    -9.693, E3 -178407.581}
SPL {X  -159.986, Y  +381.420, Z    +0.000, E1    -2.704, E3 -178408.146}
SPL {X  -159.990, Y  +385.016, Z    +0.000, E1    +0.442, E3 -178408.213}
SPL {X  -159.990, Y  +389.230, Z    +0.000, E1    +6.815, E3 -178408.348}
SPL {X  -159.990, Y  +395.332, Z    +0.000, E1   +17.451, E3 -178408.831}
SPL {X  -159.990, Y  +403.857, Z    +0.000, E1   +31.979, E3 -178410.056}
SPL {X  -159.990, Y  +416.313, Z    +0.000, E1   +46.481, E3 -178413.049}
SPL {X  -159.990, Y  +425.447, Z    +0.000, E1   +52.896, E3 -178415.957}
SPL {X  -159.990, Y  +475.808, Z    +0.000, E1   +64.751, E3 -178437.495}
SPL {X  -159.990, Y  +586.159, Z    +0.000, E1   +66.648, E3 -178516.911}
SPL {X  -159.990, Y  +602.026, Z    +0.000, E1   +66.659, E3 -178531.428}
SPL {X  -159.990, Y  +615.972, Z    +0.000, E1   +66.639, E3 -178544.256}
SPL {X  -159.990, Y  +629.811, Z    +0.000, E1   +66.653, E3 -178556.908}
SPL {X  -159.990, Y  +646.024, Z    +0.000, E1   +66.650, E3 -178571.784}
SPL {X  -159.990, Y  +658.527, Z    +0.000, E1   +66.634, E3 -178583.266}
SPL {X  -159.990, Y  +671.049, Z    +0.000, E1   +66.648, E3 -178594.715}
SPL {X  -159.230, Y  +687.071, Z    +0.000, E1   +66.569, E3 -178610.156}
SPL {X  -157.779, Y  +698.005, Z    +0.000, E1   +66.341, E3 -178621.775}
SPL {X  -156.148, Y  +706.350, Z    +0.000, E1   +66.133, E3 -178631.098}
SPL {X  -154.052, Y  +714.685, Z    +0.000, E1   +65.842, E3 -178640.885}
SPL {X  -151.381, Y  +723.275, Z    +0.000, E1   +65.482, E3 -178651.432}
SPL {X  -147.622, Y  +733.180, Z    +0.000, E1   +64.943, E3 -178664.236}
SPL {X  -144.546, Y  +740.079, Z    +0.000, E1   +64.439, E3 -178673.564}
SPL {X  -142.587, Y  +744.066, Z    +0.000, E1   +64.133, E3 -178679.058}
SPL {X  -139.326, Y  +750.145, Z    +0.000, E1   +63.650, E3 -178687.551}
SPL {X  -135.791, Y  +756.103, Z    +0.000, E1   +63.018, E3 -178696.196}
SPL {X  -133.172, Y  +760.168, Z    +0.000, E1   +62.565, E3 -178702.121}
SPL {X  -130.070, Y  +764.659, Z    +0.000, E1   +62.024, E3 -178708.717}
SPL {X  -103.420, Y  +793.570, Z    +0.000, E1   +51.337, E3 -178838.616}
ENDSPLINE

SPLINE
SPL {X  -132.256, Y  +761.529, Z    +0.000, E1   +44.935, E3 -178944.706}
SPL {X  -148.790, Y  +730.309, Z    +0.000, E1   +35.907, E3 -178965.980}
SPL {X  -157.132, Y  +701.603, Z    +0.000, E1   +22.438, E3 -178975.241}
SPL {X  -159.426, Y  +684.927, Z    +0.000, E1   +11.876, E3 -178977.860}
SPL {X  -159.929, Y  +675.915, Z    +0.000, E1    +5.290, E3 -178978.570}
SPL {X  -159.990, Y  +669.794, Z    +0.000, E1    +0.371, E3 -178978.744}
SPL {X  -159.990, Y  +668.338, Z    +0.000, E1    -1.468, E3 -178978.760}
SPL {X  -159.990, Y  +665.597, Z    +0.000, E1    -5.793, E3 -178978.839}
SPL {X  -159.990, Y  +662.769, Z    +0.000, E1   -10.720, E3 -178978.990}
SPL {X  -159.990, Y  +658.787, Z    +0.000, E1   -17.995, E3 -178979.318}
SPL {X  -159.990, Y  +653.215, Z    +0.000, E1   -27.908, E3 -178980.010}
SPL {X  -159.990, Y  +646.194, Z    +0.000, E1   -38.517, E3 -178981.299}
SPL {X  -159.990, Y  +636.314, Z    +0.000, E1   -48.490, E3 -178983.937}
SPL {X  -159.990, Y  +588.081, Z    +0.000, E1   -63.406, E3 -179005.118}
SPL {X  -159.990, Y  +471.514, Z    +0.000, E1   -66.231, E3 -179088.626}
SPL {X  -159.990, Y  +458.012, Z    +0.000, E1   -66.224, E3 -179101.256}
SPL {X  -159.990, Y  +445.900, Z    +0.000, E1   -66.225, E3 -179112.569}
ENDSPLINE

SPLINE
SPL {X  -159.990, Y  +465.730, Z    +0.000, E1   -61.693, E3 -179126.393}
ENDSPLINE

SPLINE
SPL {X  -159.990, Y  +446.910, Z    +0.000, E1   -62.394, E3 -179142.613}
SPL {X  -159.990, Y  +430.868, Z    +0.000, E1   -63.135, E3 -179154.653}
SPL {X  -159.990, Y  +416.857, Z    +0.000, E1   -63.835, E3 -179164.320}
SPL {X  -159.990, Y  +397.192, Z    +0.000, E1   -64.622, E3 -179178.613}
SPL {X  -159.570, Y  +370.917, Z    +0.000, E1   -65.713, E3 -179195.970}
SPL {X  -156.693, Y  +350.188, Z    +0.000, E1   -66.345, E3 -179210.342}
SPL {X  -153.533, Y  +337.508, Z    +0.000, E1   -66.008, E3 -179224.474}
SPL {X  -150.132, Y  +327.208, Z    +0.000, E1   -65.515, E3 -179237.260}
SPL {X  -147.311, Y  +320.081, Z    +0.000, E1   -65.083, E3 -179246.541}
SPL {X  -144.181, Y  +313.155, Z    +0.000, E1   -64.628, E3 -179255.802}
SPL {X  -141.300, Y  +307.460, Z    +0.000, E1   -64.150, E3 -179263.694}
SPL {X  -138.693, Y  +302.744, Z    +0.000, E1   -63.741, E3 -179270.308}
SPL {X  -135.031, Y  +296.690, Z    +0.000, E1   -63.147, E3 -179278.969}
SPL {X  -130.494, Y  +289.936, Z    +0.000, E1   -62.364, E3 -179288.807}
SPL {X  -102.192, Y  +259.400, Z    +0.000, E1   -52.167, E3 -179407.531}
ENDSPLINE

SPLINE
SPL {X  -140.725, Y  +306.386, Z    +0.000, E1   -41.058, E3 -179532.426}
SPL {X  -153.851, Y  +338.606, Z    +0.000, E1   -29.149, E3 -179549.043}
SPL {X  -158.264, Y  +359.064, Z    +0.000, E1   -18.155, E3 -179553.994}
SPL {X  -159.843, Y  +375.639, Z    +0.000, E1    -7.133, E3 -179556.000}
SPL {X  -159.990, Y  +384.776, Z    +0.000, E1    +0.076, E3 -179556.358}
SPL {X  -159.990, Y  +389.230, Z    +0.000, E1    +6.815, E3 -179556.497}
SPL {X  -159.990, Y  +393.768, Z    +0.000, E1   +14.836, E3 -179556.815}
SPL {X  -159.990, Y  +397.827, Z    +0.000, E1   +22.184, E3 -179557.240}
SPL {X  -159.990, Y  +403.857, Z    +0.000, E1   +31.979, E3 -179558.204}
SPL {X  -159.990, Y  +417.858, Z    +0.000, E1   +47.695, E3 -179561.690}
SPL {X  -159.990, Y  +475.808, Z    +0.000, E1   +64.751, E3 -179585.643}
SPL {X  -159.990, Y  +586.159, Z    +0.000, E1   +66.648, E3 -179665.059}
SPL {X  -159.990, Y  +602.026, Z    +0.000, E1   +66.659, E3 -179679.576}
SPL {X  -159.990, Y  +620.525, Z    +0.000, E1   +66.669, E3 -179696.513}
SPL {X  -159.990, Y  +638.202, Z    +0.000, E1   +66.649, E3 -179712.763}
SPL {X  -159.990, Y  +649.814, Z    +0.000, E1   +66.629, E3 -179723.451}
SPL {X  -159.990, Y  +658.527, Z    +0.000, E1   +66.634, E3 -179731.414}
SPL {X  -159.990, Y  +671.049, Z    +0.000, E1   +66.648, E3 -179742.863}
SPL {X  -159.230, Y  +687.071, Z    +0.000, E1   +66.569, E3 -179758.304}
SPL {X  -157.279, Y  +700.830, Z    +0.000, E1   +66.296, E3 -179772.994}
SPL {X  -154.589, Y  +712.719, Z    +0.000, E1   +65.941, E3 -179786.637}
SPL {X  -151.381, Y  +723.275, Z    +0.000, E1   +65.482, E3 -179799.580}
SPL {X  -147.622, Y  +733.180, Z    +0.000, E1   +64.943, E3 -179812.384}
SPL {X  -143.550, Y  +742.141, Z    +0.000, E1   +64.312, E3 -179824.498}
SPL {X  -140.309, Y  +748.378, Z    +0.000, E1   +63.779, E3 -179833.231}
SPL {X  -136.621, Y  +754.755, Z    +0.000, E1   +63.190, E3 -179842.348}
SPL {X  -133.172, Y  +760.168, Z    +0.000, E1   +62.565, E3 -179850.269}
SPL {X  -130.070, Y  +764.659, Z    +0.000, E1   +62.024, E3 -179856.865}
SPL {X  -103.420, Y  +793.570, Z    +0.000, E1   +51.337, E3 -179986.765}
ENDSPLINE

SPLINE
SPL {X  -141.359, Y  +746.429, Z    +0.000, E1   +41.207, E3 -180104.978}
SPL {X  -153.791, Y  +715.605, Z    +0.000, E1   +29.700, E3 -180119.748}
SPL {X  -157.923, Y  +697.131, Z    +0.000, E1   +19.758, E3 -180124.279}
SPL {X  -159.426, Y  +684.927, Z    +0.000, E1   +11.876, E3 -180126.008}
SPL {X  -159.972, Y  +673.894, Z    +0.000, E1    +3.783, E3 -180126.796}
SPL {X  -159.990, Y  +669.561, Z    +0.000, E1    +0.077, E3 -180126.894}
SPL {X  -159.990, Y  +668.338, Z    +0.000, E1    -1.468, E3 -180126.908}
SPL {X  -159.990, Y  +664.217, Z    +0.000, E1    -7.944, E3 -180127.061}
SPL {X  -159.990, Y  +658.787, Z    +0.000, E1   -17.995, E3 -180127.466}
SPL {X  -159.990, Y  +653.215, Z    +0.000, E1   -27.908, E3 -180128.158}
SPL {X  -159.990, Y  +646.194, Z    +0.000, E1   -38.517, E3 -180129.447}
SPL {X  -159.990, Y  +636.314, Z    +0.000, E1   -48.490, E3 -180132.085}
SPL {X  -159.990, Y  +588.081, Z    +0.000, E1   -63.406, E3 -180153.266}
SPL {X  -159.990, Y  +471.514, Z    +0.000, E1   -66.231, E3 -180236.774}
SPL {X  -159.990, Y  +458.012, Z    +0.000, E1   -66.224, E3 -180249.404}
SPL {X  -159.990, Y  +445.900, Z    +0.000, E1   -66.225, E3 -180260.717}
ENDSPLINE

SPLINE
SPL {X  -159.990, Y  +465.730, Z    +0.000, E1   -61.693, E3 -180274.542}
ENDSPLINE

SPLINE
SPL {X  -159.990, Y  +452.456, Z    +0.000, E1   -62.114, E3 -180286.469}
SPL {X  -159.990, Y  +436.367, Z    +0.000, E1   -62.893, E3 -180298.729}
SPL {X  -159.990, Y  +416.857, Z    +0.000, E1   -63.835, E3 -180312.468}
SPL {X  -159.990, Y  +402.942, Z    +0.000, E1   -64.377, E3 -180322.697}
SPL {X  -159.990, Y  +382.745, Z    +0.000, E1   -65.209, E3 -180336.611}
SPL {X  -158.342, Y  +359.598, Z    +0.000, E1   -66.150, E3 -180351.315}
SPL {X  -155.453, Y  +344.669, Z    +0.000, E1   -66.270, E3 -180364.157}
SPL {X  -151.958, Y  +332.444, Z    +0.000, E1   -65.791, E3 -180378.807}
SPL {X  -148.012, Y  +321.760, Z    +0.000, E1   -65.212, E3 -180392.441}
SPL {X  -144.181, Y  +313.155, Z    +0.000, E1   -64.628, E3 -180403.950}
SPL {X  -141.300, Y  +307.460, Z    +0.000, E1   -64.150, E3 -180411.842}
SPL {X  -138.693, Y  +302.744, Z    +0.000, E1   -63.741, E3 -180418.456}
SPL {X  -135.031, Y  +296.690, Z    +0.000, E1   -63.147, E3 -180427.117}
SPL {X  -130.494, Y  +289.936, Z    +0.000, E1   -62.364, E3 -180436.955}
SPL {X  -102.192, Y  +259.400, Z    +0.000, E1   -52.167, E3 -180555.680}
ENDSPLINE

SPLINE
SPL {X  -140.725, Y  +306.386, Z    +0.000, E1   -41.058, E3 -180680.574}
SPL {X  -153.851, Y  +338.606, Z    +0.000, E1   -29.149, E3 -180697.191}
SPL {X  -158.264, Y  +359.064, Z    +0.000, E1   -18.155, E3 -180702.142}
SPL {X  -159.641, Y  +371.933, Z    +0.000, E1    -9.693, E3 -180703.877}
SPL {X  -159.986, Y  +381.420, Z    +0.000, E1    -2.704, E3 -180704.442}
SPL {X  -159.990, Y  +384.527, Z    +0.000, E1    +0.013, E3 -180704.503}
SPL {X  -159.990, Y  +386.984, Z    +0.000, E1    +3.187, E3 -180704.554}
SPL {X  -159.990, Y  +392.544, Z    +0.000, E1   +12.471, E3 -180704.868}
SPL {X  -159.990, Y  +397.827, Z    +0.000, E1   +22.184, E3 -180705.389}
SPL {X  -159.990, Y  +403.857, Z    +0.000, E1   +31.979, E3 -180706.353}
SPL {X  -159.990, Y  +417.858, Z    +0.000, E1   +47.695, E3 -180709.838}
SPL {X  -159.990, Y  +475.808, Z    +0.000, E1   +64.751, E3 -180733.791}
SPL {X  -159.990, Y  +590.266, Z    +0.000, E1   +66.680, E3 -180816.909}
SPL {X  -159.990, Y  +611.678, Z    +0.000, E1   +66.672, E3 -180836.548}
SPL {X  -159.990, Y  +625.813, Z    +0.000, E1   +66.632, E3 -180849.580}
SPL {X  -159.990, Y  +638.202, Z    +0.000, E1   +66.649, E3 -180860.911}
SPL {X  -159.990, Y  +654.774, Z    +0.000, E1   +66.658, E3 -180876.080}
SPL {X  -159.990, Y  +671.049, Z    +0.000, E1   +66.648, E3 -180891.011}
SPL {X  -159.230, Y  +687.071, Z    +0.000, E1   +66.569, E3 -180906.453}
SPL {X  -157.279, Y  +700.830, Z    +0.000, E1   +66.296, E3 -180921.142}
SPL {X  -154.589, Y  +712.719, Z    +0.000, E1   +65.941, E3 -180934.785}
SPL {X  -151.381, Y  +723.275, Z    +0.000, E1   +65.482, E3 -180947.728}
SPL {X  -147.622, Y  +733.180, Z    +0.000, E1   +64.943, E3 -180960.532}
SPL {X  -143.550, Y  +742.141, Z    +0.000, E1   +64.312, E3 -180972.646}
SPL {X  -139.326, Y  +750.145, Z    +0.000, E1   +63.650, E3 -180983.847}
SPL {X  -135.791, Y  +756.103, Z    +0.000, E1   +63.018, E3 -180992.493}
SPL {X  -133.172, Y  +760.168, Z    +0.000, E1   +62.565, E3 -180998.417}
SPL {X  -130.070, Y  +764.659, Z    +0.000, E1   +62.024, E3 -181005.013}
SPL {X  -103.420, Y  +793.570, Z    +0.000, E1   +51.337, E3 -181134.913}
ENDSPLINE

SPLINE
SPL {X  -141.359, Y  +746.429, Z    +0.000, E1   +41.207, E3 -181253.127}
SPL {X  -153.791, Y  +715.605, Z    +0.000, E1   +29.700, E3 -181267.896}
SPL {X  -157.923, Y  +697.131, Z    +0.000, E1   +19.758, E3 -181272.427}
SPL {X  -159.426, Y  +684.927, Z    +0.000, E1   +11.876, E3 -181274.156}
SPL {X  -159.972, Y  +673.894, Z    +0.000, E1    +3.783, E3 -181274.944}
SPL {X  -159.990, Y  +669.561, Z    +0.000, E1    +0.077, E3 -181275.043}
SPL {X  -159.990, Y  +668.338, Z    +0.000, E1    -1.468, E3 -181275.056}
SPL {X  -159.990, Y  +664.217, Z    +0.000, E1    -7.944, E3 -181275.209}
SPL {X  -159.990, Y  +658.787, Z    +0.000, E1   -17.995, E3 -181275.614}
SPL {X  -159.990, Y  +653.215, Z    +0.000, E1   -27.908, E3 -181276.306}
SPL {X  -159.990, Y  +646.194, Z    +0.000, E1   -38.517, E3 -181277.595}
SPL {X  -159.990, Y  +636.314, Z    +0.000, E1   -48.490, E3 -181280.233}
SPL {X  -159.990, Y  +588.081, Z    +0.000, E1   -63.406, E3 -181301.414}
SPL {X  -159.990, Y  +471.514, Z    +0.000, E1   -66.231, E3 -181384.922}
SPL {X  -159.990, Y  +458.012, Z    +0.000, E1   -66.224, E3 -181397.552}
SPL {X  -159.990, Y  +445.900, Z    +0.000, E1   -66.225, E3 -181408.865}
ENDSPLINE

SPLINE
SPL {X  -159.990, Y  +465.730, Z    +0.000, E1   -61.693, E3 -181422.690}
ENDSPLINE

SPLINE
SPL {X  -159.990, Y  +446.910, Z    +0.000, E1   -62.394, E3 -181438.909}
SPL {X  -159.990, Y  +430.868, Z    +0.000, E1   -63.135, E3 -181450.949}
SPL {X  -159.990, Y  +416.857, Z    +0.000, E1   -63.835, E3 -181460.616}
SPL {X  -159.990, Y  +397.192, Z    +0.000, E1   -64.622, E3 -181474.909}
SPL {X  -159.570, Y  +370.917, Z    +0.000, E1   -65.713, E3 -181492.266}
SPL {X  -156.693, Y  +350.188, Z    +0.000, E1   -66.345, E3 -181506.638}
SPL {X  -153.533, Y  +337.508, Z    +0.000, E1   -66.008, E3 -181520.770}
SPL {X  -150.132, Y  +327.208, Z    +0.000, E1   -65.515, E3 -181533.556}
SPL {X  -146.325, Y  +317.802, Z    +0.000, E1   -64.967, E3 -181545.811}
SPL {X  -142.205, Y  +309.188, Z    +0.000, E1   -64.322, E3 -181557.547}
SPL {X  -138.693, Y  +302.744, Z    +0.000, E1   -63.741, E3 -181566.604}
SPL {X  -135.031, Y  +296.690, Z    +0.000, E1   -63.147, E3 -181575.266}
SPL {X  -130.494, Y  +289.936, Z    +0.000, E1   -62.364, E3 -181585.103}
SPL {X  -102.192, Y  +259.400, Z    +0.000, E1   -52.167, E3 -181703.828}
ENDSPLINE

SPLINE
SPL {X  -140.725, Y  +306.386, Z    +0.000, E1   -41.058, E3 -181828.722}
SPL {X  -153.851, Y  +338.606, Z    +0.000, E1   -29.149, E3 -181845.339}
SPL {X  -158.264, Y  +359.064, Z    +0.000, E1   -18.155, E3 -181850.290}
SPL {X  -159.641, Y  +371.933, Z    +0.000, E1    -9.693, E3 -181852.025}
SPL {X  -159.986, Y  +381.420, Z    +0.000, E1    -2.704, E3 -181852.590}
SPL {X  -159.990, Y  +384.527, Z    +0.000, E1    +0.013, E3 -181852.651}
SPL {X  -159.990, Y  +385.909, Z    +0.000, E1    +1.800, E3 -181852.668}
SPL {X  -159.990, Y  +389.230, Z    +0.000, E1    +6.815, E3 -181852.793}
SPL {X  -159.990, Y  +395.332, Z    +0.000, E1   +17.451, E3 -181853.275}
SPL {X  -159.990, Y  +403.857, Z    +0.000, E1   +31.979, E3 -181854.501}
SPL {X  -159.990, Y  +417.858, Z    +0.000, E1   +47.695, E3 -181857.986}
SPL {X  -159.990, Y  +475.808, Z    +0.000, E1   +64.751, E3 -181881.940}
SPL {X  -159.990, Y  +590.266, Z    +0.000, E1   +66.680, E3 -181965.057}
SPL {X  -159.990, Y  +611.678, Z    +0.000, E1   +66.672, E3 -181984.697}
SPL {X  -159.990, Y  +625.813, Z    +0.000, E1   +66.632, E3 -181997.728}
SPL {X  -159.990, Y  +638.202, Z    +0.000, E1   +66.649, E3 -182009.059}
SPL {X  -159.990, Y  +654.774, Z    +0.000, E1   +66.658, E3 -182024.229}
SPL {X  -159.990, Y  +671.049, Z    +0.000, E1   +66.648, E3 -182039.159}
SPL {X  -159.584, Y  +682.893, Z    +0.000, E1   +66.583, E3 -182050.457}
SPL {X  -158.332, Y  +694.472, Z    +0.000, E1   +66.450, E3 -182062.331}
SPL {X  -156.148, Y  +706.350, Z    +0.000, E1   +66.133, E3 -182075.542}
SPL {X  -154.052, Y  +714.685, Z    +0.000, E1   +65.842, E3 -182085.329}
SPL {X  -151.974, Y  +721.507, Z    +0.000, E1   +65.548, E3 -182093.686}
SPL {X  -149.510, Y  +728.452, Z    +0.000, E1   +65.197, E3 -182102.529}
SPL {X  -145.784, Y  +737.407, Z    +0.000, E1   +64.671, E3 -182114.319}
SPL {X  -141.166, Y  +746.792, Z    +0.000, E1   +63.950, E3 -182127.249}
SPL {X  -136.621, Y  +754.755, Z    +0.000, E1   +63.190, E3 -182138.644}
SPL {X  -133.172, Y  +760.168, Z    +0.000, E1   +62.565, E3 -182146.566}
SPL {X  -130.070, Y  +764.659, Z    +0.000, E1   +62.024, E3 -182153.161}
SPL {X  -103.420, Y  +793.570, Z    +0.000, E1   +51.337, E3 -182283.061}
ENDSPLINE

SPLINE
SPL {X  -132.256, Y  +761.529, Z    +0.000, E1   +44.935, E3 -182389.150}
SPL {X  -148.790, Y  +730.309, Z    +0.000, E1   +35.907, E3 -182410.424}
SPL {X  -157.132, Y  +701.603, Z    +0.000, E1   +22.438, E3 -182419.685}
SPL {X  -159.426, Y  +684.927, Z    +0.000, E1   +11.876, E3 -182422.304}
SPL {X  -159.929, Y  +675.915, Z    +0.000, E1    +5.290, E3 -182423.014}
SPL {X  -159.990, Y  +669.794, Z    +0.000, E1    +0.371, E3 -182423.188}
SPL {X  -159.990, Y  +668.338, Z    +0.000, E1    -1.468, E3 -182423.205}
SPL {X  -159.990, Y  +665.597, Z    +0.000, E1    -5.793, E3 -182423.283}
SPL {X  -159.990, Y  +662.769, Z    +0.000, E1   -10.720, E3 -182423.434}
SPL {X  -159.990, Y  +658.787, Z    +0.000, E1   -17.995, E3 -182423.762}
SPL {X  -159.990, Y  +653.215, Z    +0.000, E1   -27.908, E3 -182424.454}
SPL {X  -159.990, Y  +646.194, Z    +0.000, E1   -38.517, E3 -182425.743}
SPL {X  -159.990, Y  +636.314, Z    +0.000, E1   -48.490, E3 -182428.381}
SPL {X  -159.990, Y  +588.081, Z    +0.000, E1   -63.406, E3 -182449.562}
SPL {X  -159.990, Y  +471.514, Z    +0.000, E1   -66.231, E3 -182533.070}
SPL {X  -159.990, Y  +458.012, Z    +0.000, E1   -66.224, E3 -182545.700}
SPL {X  -159.990, Y  +445.900, Z    +0.000, E1   -66.225, E3 -182557.013}
ENDSPLINE

SPLINE
SPL {X  -159.990, Y  +465.730, Z    +0.000, E1   -61.693, E3 -182570.838}
ENDSPLINE

SPLINE
SPL {X  -159.990, Y  +452.456, Z    +0.000, E1   -62.114, E3 -182582.765}
SPL {X  -159.990, Y  +436.367, Z    +0.000, E1   -62.893, E3 -182595.025}
SPL {X  -159.990, Y  +416.857, Z    +0.000, E1   -63.835, E3 -182608.764}
SPL {X  -159.990, Y  +397.192, Z    +0.000, E1   -64.622, E3 -182623.057}
SPL {X  -159.902, Y  +377.209, Z    +0.000, E1   -65.412, E3 -182636.621}
SPL {X  -158.342, Y  +359.598, Z    +0.000, E1   -66.150, E3 -182647.612}
SPL {X  -155.453, Y  +344.669, Z    +0.000, E1   -66.270, E3 -182660.454}
SPL {X  -152.827, Y  +335.165, Z    +0.000, E1   -65.880, E3 -182671.811}
SPL {X  -150.132, Y  +327.208, Z    +0.000, E1   -65.515, E3 -182681.704}
SPL {X  -147.311, Y  +320.081, Z    +0.000, E1   -65.083, E3 -182690.985}
SPL {X  -144.181, Y  +313.155, Z    +0.000, E1   -64.628, E3 -182700.246}
SPL {X  -141.300, Y  +307.460, Z    +0.000, E1   -64.150, E3 -182708.138}
SPL {X  -138.693, Y  +302.744, Z    +0.000, E1   -63.741, E3 -182714.752}
SPL {X  -135.031, Y  +296.690, Z    +0.000, E1   -63.147, E3 -182723.414}
SPL {X  -130.494, Y  +289.936, Z    +0.000, E1   -62.364, E3 -182733.252}
SPL {X  -102.192, Y  +259.400, Z    +0.000, E1   -52.167, E3 -182851.976}
ENDSPLINE

SPLINE
SPL {X  -140.725, Y  +306.386, Z    +0.000, E1   -41.058, E3 -182976.870}
SPL {X  -153.851, Y  +338.606, Z    +0.000, E1   -29.149, E3 -182993.487}
SPL {X  -157.523, Y  +354.512, Z    +0.000, E1   -20.811, E3 -182997.614}
SPL {X  -159.458, Y  +369.460, Z    +0.000, E1   -11.469, E3 -182999.903}
SPL {X  -159.948, Y  +378.818, Z    +0.000, E1    -4.641, E3 -183000.649}
SPL {X  -159.990, Y  +384.776, Z    +0.000, E1    +0.076, E3 -183000.803}
SPL {X  -159.990, Y  +389.230, Z    +0.000, E1    +6.815, E3 -183000.941}
SPL {X  -159.990, Y  +393.768, Z    +0.000, E1   +14.836, E3 -183001.260}
SPL {X  -159.990, Y  +397.827, Z    +0.000, E1   +22.184, E3 -183001.685}
SPL {X  -159.990, Y  +403.857, Z    +0.000, E1   +31.979, E3 -183002.649}
SPL {X  -159.990, Y  +417.858, Z    +0.000, E1   +47.695, E3 -183006.134}
SPL {X  -159.990, Y  +475.808, Z    +0.000, E1   +64.751, E3 -183030.088}
SPL {X  -159.990, Y  +590.266, Z    +0.000, E1   +66.680, E3 -183113.205}
SPL {X  -159.990, Y  +605.903, Z    +0.000, E1   +66.635, E3 -183127.624}
SPL {X  -159.990, Y  +620.525, Z    +0.000, E1   +66.669, E3 -183140.958}
SPL {X  -159.990, Y  +638.202, Z    +0.000, E1   +66.649, E3 -183157.208}
SPL {X  -159.990, Y  +654.774, Z    +0.000, E1   +66.658, E3 -183172.377}
SPL {X  -159.990, Y  +671.049, Z    +0.000, E1   +66.648, E3 -183187.307}
SPL {X  -159.584, Y  +682.893, Z    +0.000, E1   +66.583, E3 -183198.605}
SPL {X  -158.332, Y  +694.472, Z    +0.000, E1   +66.450, E3 -183210.479}
SPL {X  -156.148, Y  +706.350, Z    +0.000, E1   +66.133, E3 -183223.690}
SPL {X  -154.052, Y  +714.685, Z    +0.000, E1   +65.842, E3 -183233.477}
SPL {X  -151.974, Y  +721.507, Z    +0.000, E1   +65.548, E3 -183241.834}
SPL {X  -149.510, Y  +728.452, Z    +0.000, E1   +65.197, E3 -183250.677}
SPL {X  -145.784, Y  +737.407, Z    +0.000, E1   +64.671, E3 -183262.468}
SPL {X  -142.587, Y  +744.066, Z    +0.000, E1   +64.133, E3 -183271.650}
SPL {X  -139.326, Y  +750.145, Z    +0.000, E1   +63.650, E3 -183280.144}
SPL {X  -135.791, Y  +756.103, Z    +0.000, E1   +63.018, E3 -183288.789}
SPL {X  -133.172, Y  +760.168, Z    +0.000, E1   +62.565, E3 -183294.714}
SPL {X  -130.070, Y  +764.659, Z    +0.000, E1   +62.024, E3 -183301.309}
SPL {X  -103.420, Y  +793.570, Z    +0.000, E1   +51.337, E3 -183431.209}
ENDSPLINE

SPLINE
SPL {X  -132.256, Y  +761.529, Z    +0.000, E1   +44.935, E3 -183537.299}
SPL {X  -148.790, Y  +730.309, Z    +0.000, E1   +35.907, E3 -183558.572}
SPL {X  -157.132, Y  +701.603, Z    +0.000, E1   +22.438, E3 -183567.833}
SPL {X  -159.426, Y  +684.927, Z    +0.000, E1   +11.876, E3 -183570.452}
SPL {X  -159.929, Y  +675.915, Z    +0.000, E1    +5.290, E3 -183571.163}
SPL {X  -159.990, Y  +669.794, Z    +0.000, E1    +0.371, E3 -183571.336}
SPL {X  -159.990, Y  +668.338, Z    +0.000, E1    -1.468, E3 -183571.353}
SPL {X  -159.990, Y  +664.217, Z    +0.000, E1    -7.944, E3 -183571.505}
SPL {X  -159.990, Y  +657.963, Z    +0.000, E1   -19.417, E3 -183572.002}
SPL {X  -159.990, Y  +649.570, Z    +0.000, E1   -33.681, E3 -183573.226}
SPL {X  -159.990, Y  +636.314, Z    +0.000, E1   -48.490, E3 -183576.529}
SPL {X  -159.990, Y  +588.081, Z    +0.000, E1   -63.406, E3 -183597.711}
SPL {X  -159.990, Y  +471.514, Z    +0.000, E1   -66.231, E3 -183681.219}
SPL {X  -159.990, Y  +458.012, Z    +0.000, E1   -66.224, E3 -183693.848}
SPL {X  -159.990, Y  +445.900, Z    +0.000, E1   -66.225, E3 -183705.161}
ENDSPLINE

SPLINE
SPL {X  -159.990, Y  +465.730, Z    +0.000, E1   -61.693, E3 -183718.986}
ENDSPLINE

SPLINE
SPL {X  -159.990, Y  +446.910, Z    +0.000, E1   -62.394, E3 -183735.205}
SPL {X  -159.990, Y  +430.868, Z    +0.000, E1   -63.135, E3 -183747.245}
SPL {X  -159.990, Y  +416.857, Z    +0.000, E1   -63.835, E3 -183756.912}
SPL {X  -159.990, Y  +397.192, Z    +0.000, E1   -64.622, E3 -183771.205}
SPL {X  -159.902, Y  +377.209, Z    +0.000, E1   -65.412, E3 -183784.769}
SPL {X  -158.342, Y  +359.598, Z    +0.000, E1   -66.150, E3 -183795.760}
SPL {X  -155.453, Y  +344.669, Z    +0.000, E1   -66.270, E3 -183808.602}
SPL {X  -152.827, Y  +335.165, Z    +0.000, E1   -65.880, E3 -183819.960}
SPL {X  -150.132, Y  +327.208, Z    +0.000, E1   -65.515, E3 -183829.852}
SPL {X  -147.311, Y  +320.081, Z    +0.000, E1   -65.083, E3 -183839.133}
SPL {X  -144.181, Y  +313.155, Z    +0.000, E1   -64.628, E3 -183848.395}
SPL {X  -141.300, Y  +307.460, Z    +0.000, E1   -64.150, E3 -183856.286}
SPL {X  -138.693, Y  +302.744, Z    +0.000, E1   -63.741, E3 -183862.900}
SPL {X  -135.977, Y  +298.197, Z    +0.000, E1   -63.280, E3 -183869.420}
SPL {X  -132.828, Y  +293.318, Z    +0.000, E1   -62.759, E3 -183876.474}
SPL {X  -129.451, Y  +288.482, Z    +0.000, E1   -62.137, E3 -183883.577}
SPL {X  -102.192, Y  +259.400, Z    +0.000, E1   -52.167, E3 -184000.124}
ENDSPLINE

SPLINE
SPL {X  -140.725, Y  +306.386, Z    +0.000, E1   -41.058, E3 -184125.018}
SPL {X  -153.851, Y  +338.606, Z    +0.000, E1   -29.149, E3 -184141.635}
SPL {X  -158.264, Y  +359.064, Z    +0.000, E1   -18.155, E3 -184146.586}
SPL {X  -159.843, Y  +375.639, Z    +0.000, E1    -7.133, E3 -184148.593}
SPL {X  -159.990, Y  +384.256, Z    +0.000, E1    -0.337, E3 -184148.944}
SPL {X  -159.990, Y  +386.984, Z    +0.000, E1    +3.187, E3 -184148.999}
SPL {X  -159.990, Y  +390.572, Z    +0.000, E1    +9.243, E3 -184149.158}
SPL {X  -159.990, Y  +395.332, Z    +0.000, E1   +17.451, E3 -184149.572}
SPL {X  -159.990, Y  +403.857, Z    +0.000, E1   +31.979, E3 -184150.797}
SPL {X  -159.990, Y  +417.858, Z    +0.000, E1   +47.695, E3 -184154.282}
SPL {X  -159.990, Y  +475.808, Z    +0.000, E1   +64.751, E3 -184178.236}
SPL {X  -159.990, Y  +590.266, Z    +0.000, E1   +66.680, E3 -184261.353}
SPL {X  -159.990, Y  +611.678, Z    +0.000, E1   +66.672, E3 -184280.993}
SPL {X  -159.990, Y  +629.811, Z    +0.000, E1   +66.653, E3 -184297.649}
SPL {X  -159.990, Y  +646.024, Z    +0.000, E1   +66.650, E3 -184312.525}
SPL {X  -159.990, Y  +658.527, Z    +0.000, E1   +66.634, E3 -184324.007}
SPL {X  -159.990, Y  +671.049, Z    +0.000, E1   +66.648, E3 -184335.456}
SPL {X  -159.584, Y  +682.893, Z    +0.000, E1   +66.583, E3 -184346.753}
SPL {X  -158.332, Y  +694.472, Z    +0.000, E1   +66.450, E3 -184358.627}
SPL {X  -156.148, Y  +706.350, Z    +0.000, E1   +66.133, E3 -184371.838}
SPL {X  -154.052, Y  +714.685, Z    +0.000, E1   +65.842, E3 -184381.626}
SPL {X  -151.974, Y  +721.507, Z    +0.000, E1   +65.548, E3 -184389.982}
SPL {X  -149.510, Y  +728.452, Z    +0.000, E1   +65.197, E3 -184398.825}
SPL {X  -145.784, Y  +737.407, Z    +0.000, E1   +64.671, E3 -184410.616}
SPL {X  -142.587, Y  +744.066, Z    +0.000, E1   +64.133, E3 -184419.799}
SPL {X  -139.326, Y  +750.145, Z    +0.000, E1   +63.650, E3 -184428.292}
SPL {X  -135.791, Y  +756.103, Z    +0.000, E1   +63.018, E3 -184436.937}
SPL {X  -133.172, Y  +760.168, Z    +0.000, E1   +62.565, E3 -184442.862}
SPL {X  -130.070, Y  +764.659, Z    +0.000, E1   +62.024, E3 -184449.457}
SPL {X  -103.420, Y  +793.570, Z    +0.000, E1   +51.337, E3 -184579.357}
ENDSPLINE

SPLINE
SPL {X  -132.256, Y  +761.529, Z    +0.000, E1   +44.935, E3 -184685.447}
SPL {X  -148.790, Y  +730.309, Z    +0.000, E1   +35.907, E3 -184706.720}
SPL {X  -157.132, Y  +701.603, Z    +0.000, E1   +22.438, E3 -184715.981}
SPL {X  -159.426, Y  +684.927, Z    +0.000, E1   +11.876, E3 -184718.600}
SPL {X  -159.929, Y  +675.915, Z    +0.000, E1    +5.290, E3 -184719.311}
SPL {X  -159.990, Y  +669.794, Z    +0.000, E1    +0.371, E3 -184719.484}
SPL {X  -159.990, Y  +668.338, Z    +0.000, E1    -1.468, E3 -184719.501}
SPL {X  -159.990, Y  +665.597, Z    +0.000, E1    -5.793, E3 -184719.580}
SPL {X  -159.990, Y  +662.769, Z    +0.000, E1   -10.720, E3 -184719.731}
SPL {X  -159.990, Y  +658.787, Z    +0.000, E1   -17.995, E3 -184720.059}
SPL {X  -159.990, Y  +653.215, Z    +0.000, E1   -27.908, E3 -184720.751}
SPL {X  -159.990, Y  +646.194, Z    +0.000, E1   -38.517, E3 -184722.039}
SPL {X  -159.990, Y  +636.314, Z    +0.000, E1   -48.490, E3 -184724.677}
SPL {X  -159.990, Y  +588.081, Z    +0.000, E1   -63.406, E3 -184745.859}
SPL {X  -159.990, Y  +471.514, Z    +0.000, E1   -66.231, E3 -184829.367}
SPL {X  -159.990, Y  +458.012, Z    +0.000, E1   -66.224, E3 -184841.996}
SPL {X  -159.990, Y  +445.900, Z    +0.000, E1   -66.225, E3 -184853.309}
ENDSPLINE

SPLINE
SPL {X  -159.990, Y  +468.953, Z    +0.000, E1   -61.697, E3 -184863.268}
ENDSPLINE

